Error[1164].CreateEx(TC_Events.Error.Error1164,FALSE,0);
Error[1165].CreateEx(TC_Events.Error.Error1165,FALSE,0);
Error[1166].CreateEx(TC_Events.Error.Error1166,FALSE,0);
Error[1167].CreateEx(TC_Events.Error.Error1167,FALSE,0);
Error[1168].CreateEx(TC_Events.Error.Error1168,FALSE,0);
Error[1169].CreateEx(TC_Events.Error.Error1169,FALSE,0);
Error[1170].CreateEx(TC_Events.Error.Error1170,FALSE,0);
Error[1171].CreateEx(TC_Events.Error.Error1171,FALSE,0);
Error[1172].CreateEx(TC_Events.Error.Error1172,FALSE,0);
Error[1173].CreateEx(TC_Events.Error.Error1173,FALSE,0);
Error[1174].CreateEx(TC_Events.Error.Error1174,FALSE,0);
Error[1175].CreateEx(TC_Events.Error.Error1175,FALSE,0);
Error[1176].CreateEx(TC_Events.Error.Error1176,FALSE,0);
Error[1177].CreateEx(TC_Events.Error.Error1177,FALSE,0);
Error[1178].CreateEx(TC_Events.Error.Error1178,FALSE,0);
Error[1179].CreateEx(TC_Events.Error.Error1179,FALSE,0);
Error[1180].CreateEx(TC_Events.Error.Error1180,FALSE,0);
Error[1181].CreateEx(TC_Events.Error.Error1181,FALSE,0);
Error[1182].CreateEx(TC_Events.Error.Error1182,FALSE,0);
Error[1183].CreateEx(TC_Events.Error.Error1183,FALSE,0);
Error[1184].CreateEx(TC_Events.Error.Error1184,FALSE,0);
Error[1185].CreateEx(TC_Events.Error.Error1185,FALSE,0);
Error[1186].CreateEx(TC_Events.Error.Error1186,FALSE,0);
Error[1187].CreateEx(TC_Events.Error.Error1187,FALSE,0);
Error[1188].CreateEx(TC_Events.Error.Error1188,FALSE,0);
Error[1189].CreateEx(TC_Events.Error.Error1189,FALSE,0);
Error[1190].CreateEx(TC_Events.Error.Error1190,FALSE,0);
Error[1191].CreateEx(TC_Events.Error.Error1191,FALSE,0);
Error[1192].CreateEx(TC_Events.Error.Error1192,FALSE,0);
Error[1193].CreateEx(TC_Events.Error.Error1193,FALSE,0);
Error[1194].CreateEx(TC_Events.Error.Error1194,FALSE,0);
Error[1195].CreateEx(TC_Events.Error.Error1195,FALSE,0);
Error[1196].CreateEx(TC_Events.Error.Error1196,FALSE,0);
Error[1197].CreateEx(TC_Events.Error.Error1197,FALSE,0);
Error[1198].CreateEx(TC_Events.Error.Error1198,FALSE,0);
Error[1199].CreateEx(TC_Events.Error.Error1199,FALSE,0);
Error[1200].CreateEx(TC_Events.Error.Error1200,FALSE,0);
Error[1201].CreateEx(TC_Events.Error.Error1201,FALSE,0);
Error[1202].CreateEx(TC_Events.Error.Error1202,FALSE,0);
Error[1203].CreateEx(TC_Events.Error.Error1203,FALSE,0);
Error[1204].CreateEx(TC_Events.Error.Error1204,FALSE,0);
Error[1205].CreateEx(TC_Events.Error.Error1205,FALSE,0);
Error[1206].CreateEx(TC_Events.Error.Error1206,FALSE,0);
Error[1207].CreateEx(TC_Events.Error.Error1207,FALSE,0);
Error[1208].CreateEx(TC_Events.Error.Error1208,FALSE,0);
Error[1209].CreateEx(TC_Events.Error.Error1209,FALSE,0);
Error[1210].CreateEx(TC_Events.Error.Error1210,FALSE,0);
Error[1211].CreateEx(TC_Events.Error.Error1211,FALSE,0);
Error[1212].CreateEx(TC_Events.Error.Error1212,FALSE,0);
Error[1213].CreateEx(TC_Events.Error.Error1213,FALSE,0);
Error[1214].CreateEx(TC_Events.Error.Error1214,FALSE,0);
Error[1215].CreateEx(TC_Events.Error.Error1215,FALSE,0);
Error[1216].CreateEx(TC_Events.Error.Error1216,FALSE,0);
Error[1217].CreateEx(TC_Events.Error.Error1217,FALSE,0);
Error[1218].CreateEx(TC_Events.Error.Error1218,FALSE,0);
Error[1219].CreateEx(TC_Events.Error.Error1219,FALSE,0);
Error[1220].CreateEx(TC_Events.Error.Error1220,FALSE,0);
Error[1221].CreateEx(TC_Events.Error.Error1221,FALSE,0);
Error[1222].CreateEx(TC_Events.Error.Error1222,FALSE,0);
Error[1223].CreateEx(TC_Events.Error.Error1223,FALSE,0);
Error[1224].CreateEx(TC_Events.Error.Error1224,FALSE,0);
Error[1225].CreateEx(TC_Events.Error.Error1225,FALSE,0);
Error[1226].CreateEx(TC_Events.Error.Error1226,FALSE,0);
Error[1227].CreateEx(TC_Events.Error.Error1227,FALSE,0);
Error[1228].CreateEx(TC_Events.Error.Error1228,FALSE,0);
Error[1229].CreateEx(TC_Events.Error.Error1229,FALSE,0);
Error[1230].CreateEx(TC_Events.Error.Error1230,FALSE,0);
Error[1231].CreateEx(TC_Events.Error.Error1231,FALSE,0);
Error[1232].CreateEx(TC_Events.Error.Error1232,FALSE,0);
Error[1233].CreateEx(TC_Events.Error.Error1233,FALSE,0);
Error[1234].CreateEx(TC_Events.Error.Error1234,FALSE,0);
Error[1235].CreateEx(TC_Events.Error.Error1235,FALSE,0);
Error[1236].CreateEx(TC_Events.Error.Error1236,FALSE,0);
Error[1237].CreateEx(TC_Events.Error.Error1237,FALSE,0);
Error[1238].CreateEx(TC_Events.Error.Error1238,FALSE,0);
Error[1239].CreateEx(TC_Events.Error.Error1239,FALSE,0);
Error[1240].CreateEx(TC_Events.Error.Error1240,FALSE,0);
Error[1241].CreateEx(TC_Events.Error.Error1241,FALSE,0);
Error[1242].CreateEx(TC_Events.Error.Error1242,FALSE,0);
Error[1243].CreateEx(TC_Events.Error.Error1243,FALSE,0);
Error[1244].CreateEx(TC_Events.Error.Error1244,FALSE,0);
Error[1245].CreateEx(TC_Events.Error.Error1245,FALSE,0);
Error[1246].CreateEx(TC_Events.Error.Error1246,FALSE,0);
Error[1247].CreateEx(TC_Events.Error.Error1247,FALSE,0);
Error[1248].CreateEx(TC_Events.Error.Error1248,FALSE,0);
Error[1249].CreateEx(TC_Events.Error.Error1249,FALSE,0);
Error[1250].CreateEx(TC_Events.Error.Error1250,FALSE,0);
Error[1251].CreateEx(TC_Events.Error.Error1251,FALSE,0);
Error[1252].CreateEx(TC_Events.Error.Error1252,FALSE,0);
Error[1253].CreateEx(TC_Events.Error.Error1253,FALSE,0);
Error[1254].CreateEx(TC_Events.Error.Error1254,FALSE,0);
Error[1255].CreateEx(TC_Events.Error.Error1255,FALSE,0);
Error[1256].CreateEx(TC_Events.Error.Error1256,FALSE,0);
Error[1257].CreateEx(TC_Events.Error.Error1257,FALSE,0);
Error[1258].CreateEx(TC_Events.Error.Error1258,FALSE,0);
Error[1259].CreateEx(TC_Events.Error.Error1259,FALSE,0);
Error[1260].CreateEx(TC_Events.Error.Error1260,FALSE,0);
Error[1261].CreateEx(TC_Events.Error.Error1261,FALSE,0);
Error[1262].CreateEx(TC_Events.Error.Error1262,FALSE,0);
Error[1263].CreateEx(TC_Events.Error.Error1263,FALSE,0);
Error[1264].CreateEx(TC_Events.Error.Error1264,FALSE,0);
Error[1265].CreateEx(TC_Events.Error.Error1265,FALSE,0);
Error[1266].CreateEx(TC_Events.Error.Error1266,FALSE,0);
Error[1267].CreateEx(TC_Events.Error.Error1267,FALSE,0);
Error[1268].CreateEx(TC_Events.Error.Error1268,FALSE,0);
Error[1269].CreateEx(TC_Events.Error.Error1269,FALSE,0);
Error[1270].CreateEx(TC_Events.Error.Error1270,FALSE,0);
Error[1271].CreateEx(TC_Events.Error.Error1271,FALSE,0);
Error[1272].CreateEx(TC_Events.Error.Error1272,FALSE,0);
Error[1273].CreateEx(TC_Events.Error.Error1273,FALSE,0);
Error[1274].CreateEx(TC_Events.Error.Error1274,FALSE,0);
Error[1275].CreateEx(TC_Events.Error.Error1275,FALSE,0);
Error[1276].CreateEx(TC_Events.Error.Error1276,FALSE,0);
Error[1277].CreateEx(TC_Events.Error.Error1277,FALSE,0);
Error[1278].CreateEx(TC_Events.Error.Error1278,FALSE,0);
Error[1279].CreateEx(TC_Events.Error.Error1279,FALSE,0);
Error[1280].CreateEx(TC_Events.Error.Error1280,FALSE,0);
Error[1281].CreateEx(TC_Events.Error.Error1281,FALSE,0);
Error[1282].CreateEx(TC_Events.Error.Error1282,FALSE,0);
Error[1283].CreateEx(TC_Events.Error.Error1283,FALSE,0);
Error[1284].CreateEx(TC_Events.Error.Error1284,FALSE,0);
Error[1285].CreateEx(TC_Events.Error.Error1285,FALSE,0);
Error[1286].CreateEx(TC_Events.Error.Error1286,FALSE,0);
Error[1287].CreateEx(TC_Events.Error.Error1287,FALSE,0);
Error[1288].CreateEx(TC_Events.Error.Error1288,FALSE,0);
Error[1289].CreateEx(TC_Events.Error.Error1289,FALSE,0);
Error[1290].CreateEx(TC_Events.Error.Error1290,FALSE,0);
Error[1291].CreateEx(TC_Events.Error.Error1291,FALSE,0);
Error[1292].CreateEx(TC_Events.Error.Error1292,FALSE,0);
Error[1293].CreateEx(TC_Events.Error.Error1293,FALSE,0);
Error[1294].CreateEx(TC_Events.Error.Error1294,FALSE,0);
Error[1295].CreateEx(TC_Events.Error.Error1295,FALSE,0);
Error[1296].CreateEx(TC_Events.Error.Error1296,FALSE,0);
Error[1297].CreateEx(TC_Events.Error.Error1297,FALSE,0);
Error[1298].CreateEx(TC_Events.Error.Error1298,FALSE,0);
Error[1299].CreateEx(TC_Events.Error.Error1299,FALSE,0);
Error[1300].CreateEx(TC_Events.Error.Error1300,FALSE,0);
Error[1301].CreateEx(TC_Events.Error.Error1301,FALSE,0);
Error[1302].CreateEx(TC_Events.Error.Error1302,FALSE,0);
Error[1303].CreateEx(TC_Events.Error.Error1303,FALSE,0);
Error[1304].CreateEx(TC_Events.Error.Error1304,FALSE,0);
Error[1305].CreateEx(TC_Events.Error.Error1305,FALSE,0);
Error[1306].CreateEx(TC_Events.Error.Error1306,FALSE,0);
Error[1307].CreateEx(TC_Events.Error.Error1307,FALSE,0);
Error[1308].CreateEx(TC_Events.Error.Error1308,FALSE,0);
Error[1309].CreateEx(TC_Events.Error.Error1309,FALSE,0);
Error[1310].CreateEx(TC_Events.Error.Error1310,FALSE,0);
Error[1311].CreateEx(TC_Events.Error.Error1311,FALSE,0);
Error[1312].CreateEx(TC_Events.Error.Error1312,FALSE,0);
Error[1313].CreateEx(TC_Events.Error.Error1313,FALSE,0);
Error[1314].CreateEx(TC_Events.Error.Error1314,FALSE,0);
Error[1315].CreateEx(TC_Events.Error.Error1315,FALSE,0);
Error[1316].CreateEx(TC_Events.Error.Error1316,FALSE,0);
Error[1317].CreateEx(TC_Events.Error.Error1317,FALSE,0);
Error[1318].CreateEx(TC_Events.Error.Error1318,FALSE,0);
Error[1319].CreateEx(TC_Events.Error.Error1319,FALSE,0);
Error[1320].CreateEx(TC_Events.Error.Error1320,FALSE,0);
Error[1321].CreateEx(TC_Events.Error.Error1321,FALSE,0);
Error[1322].CreateEx(TC_Events.Error.Error1322,FALSE,0);
Error[1323].CreateEx(TC_Events.Error.Error1323,FALSE,0);
Error[1324].CreateEx(TC_Events.Error.Error1324,FALSE,0);
Error[1325].CreateEx(TC_Events.Error.Error1325,FALSE,0);
Error[1326].CreateEx(TC_Events.Error.Error1326,FALSE,0);
Error[1327].CreateEx(TC_Events.Error.Error1327,FALSE,0);
Error[1328].CreateEx(TC_Events.Error.Error1328,FALSE,0);
Error[1329].CreateEx(TC_Events.Error.Error1329,FALSE,0);
Error[1330].CreateEx(TC_Events.Error.Error1330,FALSE,0);
Error[1331].CreateEx(TC_Events.Error.Error1331,FALSE,0);
Error[1332].CreateEx(TC_Events.Error.Error1332,FALSE,0);
Error[1333].CreateEx(TC_Events.Error.Error1333,FALSE,0);
Error[1334].CreateEx(TC_Events.Error.Error1334,FALSE,0);
Error[1335].CreateEx(TC_Events.Error.Error1335,FALSE,0);
Error[1336].CreateEx(TC_Events.Error.Error1336,FALSE,0);
Error[1337].CreateEx(TC_Events.Error.Error1337,FALSE,0);
Error[1338].CreateEx(TC_Events.Error.Error1338,FALSE,0);
Error[1339].CreateEx(TC_Events.Error.Error1339,FALSE,0);
Error[1340].CreateEx(TC_Events.Error.Error1340,FALSE,0);
Error[1341].CreateEx(TC_Events.Error.Error1341,FALSE,0);
Error[1342].CreateEx(TC_Events.Error.Error1342,FALSE,0);
Error[1343].CreateEx(TC_Events.Error.Error1343,FALSE,0);
Error[1344].CreateEx(TC_Events.Error.Error1344,FALSE,0);
Error[1345].CreateEx(TC_Events.Error.Error1345,FALSE,0);
Error[1346].CreateEx(TC_Events.Error.Error1346,FALSE,0);
Error[1347].CreateEx(TC_Events.Error.Error1347,FALSE,0);
Error[1348].CreateEx(TC_Events.Error.Error1348,FALSE,0);
Error[1349].CreateEx(TC_Events.Error.Error1349,FALSE,0);
Error[1350].CreateEx(TC_Events.Error.Error1350,FALSE,0);
Error[1351].CreateEx(TC_Events.Error.Error1351,FALSE,0);
Error[1352].CreateEx(TC_Events.Error.Error1352,FALSE,0);
Error[1353].CreateEx(TC_Events.Error.Error1353,FALSE,0);
Error[1354].CreateEx(TC_Events.Error.Error1354,FALSE,0);
Error[1355].CreateEx(TC_Events.Error.Error1355,FALSE,0);
Error[1356].CreateEx(TC_Events.Error.Error1356,FALSE,0);
Error[1357].CreateEx(TC_Events.Error.Error1357,FALSE,0);
Error[1358].CreateEx(TC_Events.Error.Error1358,FALSE,0);
Error[1359].CreateEx(TC_Events.Error.Error1359,FALSE,0);
Error[1360].CreateEx(TC_Events.Error.Error1360,FALSE,0);
Error[1361].CreateEx(TC_Events.Error.Error1361,FALSE,0);
Error[1362].CreateEx(TC_Events.Error.Error1362,FALSE,0);
Error[1363].CreateEx(TC_Events.Error.Error1363,FALSE,0);
Error[1364].CreateEx(TC_Events.Error.Error1364,FALSE,0);
Error[1365].CreateEx(TC_Events.Error.Error1365,FALSE,0);
Error[1366].CreateEx(TC_Events.Error.Error1366,FALSE,0);
Error[1367].CreateEx(TC_Events.Error.Error1367,FALSE,0);
Error[1368].CreateEx(TC_Events.Error.Error1368,FALSE,0);
Error[1369].CreateEx(TC_Events.Error.Error1369,FALSE,0);
Error[1370].CreateEx(TC_Events.Error.Error1370,FALSE,0);
Error[1371].CreateEx(TC_Events.Error.Error1371,FALSE,0);
Error[1372].CreateEx(TC_Events.Error.Error1372,FALSE,0);
Error[1373].CreateEx(TC_Events.Error.Error1373,FALSE,0);
Error[1374].CreateEx(TC_Events.Error.Error1374,FALSE,0);
Error[1375].CreateEx(TC_Events.Error.Error1375,FALSE,0);
Error[1376].CreateEx(TC_Events.Error.Error1376,FALSE,0);
Error[1377].CreateEx(TC_Events.Error.Error1377,FALSE,0);
Error[1378].CreateEx(TC_Events.Error.Error1378,FALSE,0);
Error[1379].CreateEx(TC_Events.Error.Error1379,FALSE,0);
Error[1380].CreateEx(TC_Events.Error.Error1380,FALSE,0);
Error[1381].CreateEx(TC_Events.Error.Error1381,FALSE,0);
Error[1382].CreateEx(TC_Events.Error.Error1382,FALSE,0);
Error[1383].CreateEx(TC_Events.Error.Error1383,FALSE,0);
Error[1384].CreateEx(TC_Events.Error.Error1384,FALSE,0);
Error[1385].CreateEx(TC_Events.Error.Error1385,FALSE,0);
Error[1386].CreateEx(TC_Events.Error.Error1386,FALSE,0);
Error[1387].CreateEx(TC_Events.Error.Error1387,FALSE,0);
Error[1388].CreateEx(TC_Events.Error.Error1388,FALSE,0);
Error[1389].CreateEx(TC_Events.Error.Error1389,FALSE,0);
Error[1390].CreateEx(TC_Events.Error.Error1390,FALSE,0);
Error[1391].CreateEx(TC_Events.Error.Error1391,FALSE,0);
Error[1392].CreateEx(TC_Events.Error.Error1392,FALSE,0);
Error[1393].CreateEx(TC_Events.Error.Error1393,FALSE,0);
Error[1394].CreateEx(TC_Events.Error.Error1394,FALSE,0);
Error[1395].CreateEx(TC_Events.Error.Error1395,FALSE,0);
Error[1396].CreateEx(TC_Events.Error.Error1396,FALSE,0);
Error[1397].CreateEx(TC_Events.Error.Error1397,FALSE,0);
Error[1398].CreateEx(TC_Events.Error.Error1398,FALSE,0);
Error[1399].CreateEx(TC_Events.Error.Error1399,FALSE,0);
Error[1400].CreateEx(TC_Events.Error.Error1400,FALSE,0);
Error[1401].CreateEx(TC_Events.Error.Error1401,FALSE,0);
Error[1402].CreateEx(TC_Events.Error.Error1402,FALSE,0);
Error[1403].CreateEx(TC_Events.Error.Error1403,FALSE,0);
Error[1404].CreateEx(TC_Events.Error.Error1404,FALSE,0);
Error[1405].CreateEx(TC_Events.Error.Error1405,FALSE,0);
Error[1406].CreateEx(TC_Events.Error.Error1406,FALSE,0);
Error[1407].CreateEx(TC_Events.Error.Error1407,FALSE,0);
Error[1408].CreateEx(TC_Events.Error.Error1408,FALSE,0);
Error[1409].CreateEx(TC_Events.Error.Error1409,FALSE,0);
Error[1410].CreateEx(TC_Events.Error.Error1410,FALSE,0);
Error[1411].CreateEx(TC_Events.Error.Error1411,FALSE,0);
Error[1412].CreateEx(TC_Events.Error.Error1412,FALSE,0);
Error[1413].CreateEx(TC_Events.Error.Error1413,FALSE,0);
Error[1414].CreateEx(TC_Events.Error.Error1414,FALSE,0);
Error[1415].CreateEx(TC_Events.Error.Error1415,FALSE,0);
Error[1416].CreateEx(TC_Events.Error.Error1416,FALSE,0);
Error[1417].CreateEx(TC_Events.Error.Error1417,FALSE,0);
Error[1418].CreateEx(TC_Events.Error.Error1418,FALSE,0);
Error[1419].CreateEx(TC_Events.Error.Error1419,FALSE,0);
Error[1420].CreateEx(TC_Events.Error.Error1420,FALSE,0);
Error[1421].CreateEx(TC_Events.Error.Error1421,FALSE,0);
Error[1422].CreateEx(TC_Events.Error.Error1422,FALSE,0);
Error[1423].CreateEx(TC_Events.Error.Error1423,FALSE,0);
Error[1424].CreateEx(TC_Events.Error.Error1424,FALSE,0);
Error[1425].CreateEx(TC_Events.Error.Error1425,FALSE,0);
Error[1426].CreateEx(TC_Events.Error.Error1426,FALSE,0);
Error[1427].CreateEx(TC_Events.Error.Error1427,FALSE,0);
Error[1428].CreateEx(TC_Events.Error.Error1428,FALSE,0);
Error[1429].CreateEx(TC_Events.Error.Error1429,FALSE,0);
Error[1430].CreateEx(TC_Events.Error.Error1430,FALSE,0);
Error[1431].CreateEx(TC_Events.Error.Error1431,FALSE,0);
Error[1432].CreateEx(TC_Events.Error.Error1432,FALSE,0);
Error[1433].CreateEx(TC_Events.Error.Error1433,FALSE,0);
Error[1434].CreateEx(TC_Events.Error.Error1434,FALSE,0);
Error[1435].CreateEx(TC_Events.Error.Error1435,FALSE,0);
Error[1436].CreateEx(TC_Events.Error.Error1436,FALSE,0);
Error[1437].CreateEx(TC_Events.Error.Error1437,FALSE,0);
Error[1438].CreateEx(TC_Events.Error.Error1438,FALSE,0);
Error[1439].CreateEx(TC_Events.Error.Error1439,FALSE,0);
Error[1440].CreateEx(TC_Events.Error.Error1440,FALSE,0);
Error[1441].CreateEx(TC_Events.Error.Error1441,FALSE,0);
Error[1442].CreateEx(TC_Events.Error.Error1442,FALSE,0);
Error[1443].CreateEx(TC_Events.Error.Error1443,FALSE,0);
Error[1444].CreateEx(TC_Events.Error.Error1444,FALSE,0);
Error[1445].CreateEx(TC_Events.Error.Error1445,FALSE,0);
Error[1446].CreateEx(TC_Events.Error.Error1446,FALSE,0);
Error[1447].CreateEx(TC_Events.Error.Error1447,FALSE,0);
Error[1448].CreateEx(TC_Events.Error.Error1448,FALSE,0);
Error[1449].CreateEx(TC_Events.Error.Error1449,FALSE,0);
Error[1450].CreateEx(TC_Events.Error.Error1450,FALSE,0);
Error[1451].CreateEx(TC_Events.Error.Error1451,FALSE,0);
Error[1452].CreateEx(TC_Events.Error.Error1452,FALSE,0);
Error[1453].CreateEx(TC_Events.Error.Error1453,FALSE,0);
Error[1454].CreateEx(TC_Events.Error.Error1454,FALSE,0);
Error[1455].CreateEx(TC_Events.Error.Error1455,FALSE,0);
Error[1456].CreateEx(TC_Events.Error.Error1456,FALSE,0);
Error[1457].CreateEx(TC_Events.Error.Error1457,FALSE,0);
Error[1458].CreateEx(TC_Events.Error.Error1458,FALSE,0);
Error[1459].CreateEx(TC_Events.Error.Error1459,FALSE,0);
Error[1460].CreateEx(TC_Events.Error.Error1460,FALSE,0);
Error[1461].CreateEx(TC_Events.Error.Error1461,FALSE,0);
Error[1462].CreateEx(TC_Events.Error.Error1462,FALSE,0);
Error[1463].CreateEx(TC_Events.Error.Error1463,FALSE,0);
Error[1464].CreateEx(TC_Events.Error.Error1464,FALSE,0);
Error[1465].CreateEx(TC_Events.Error.Error1465,FALSE,0);
Error[1466].CreateEx(TC_Events.Error.Error1466,FALSE,0);
Error[1467].CreateEx(TC_Events.Error.Error1467,FALSE,0);
Error[1468].CreateEx(TC_Events.Error.Error1468,FALSE,0);
Error[1469].CreateEx(TC_Events.Error.Error1469,FALSE,0);
Error[1470].CreateEx(TC_Events.Error.Error1470,FALSE,0);
Error[1471].CreateEx(TC_Events.Error.Error1471,FALSE,0);
Error[1472].CreateEx(TC_Events.Error.Error1472,FALSE,0);
Error[1473].CreateEx(TC_Events.Error.Error1473,FALSE,0);
Error[1474].CreateEx(TC_Events.Error.Error1474,FALSE,0);
Error[1475].CreateEx(TC_Events.Error.Error1475,FALSE,0);
Error[1476].CreateEx(TC_Events.Error.Error1476,FALSE,0);
Error[1477].CreateEx(TC_Events.Error.Error1477,FALSE,0);
Error[1478].CreateEx(TC_Events.Error.Error1478,FALSE,0);
Error[1479].CreateEx(TC_Events.Error.Error1479,FALSE,0);
Error[1480].CreateEx(TC_Events.Error.Error1480,FALSE,0);
Error[1481].CreateEx(TC_Events.Error.Error1481,FALSE,0);
Error[1482].CreateEx(TC_Events.Error.Error1482,FALSE,0);
Error[1483].CreateEx(TC_Events.Error.Error1483,FALSE,0);
Error[1484].CreateEx(TC_Events.Error.Error1484,FALSE,0);
Error[1485].CreateEx(TC_Events.Error.Error1485,FALSE,0);
Error[1486].CreateEx(TC_Events.Error.Error1486,FALSE,0);
Error[1487].CreateEx(TC_Events.Error.Error1487,FALSE,0);
Error[1488].CreateEx(TC_Events.Error.Error1488,FALSE,0);
Error[1489].CreateEx(TC_Events.Error.Error1489,FALSE,0);
Error[1490].CreateEx(TC_Events.Error.Error1490,FALSE,0);
Error[1491].CreateEx(TC_Events.Error.Error1491,FALSE,0);
Error[1492].CreateEx(TC_Events.Error.Error1492,FALSE,0);
Error[1493].CreateEx(TC_Events.Error.Error1493,FALSE,0);
Error[1494].CreateEx(TC_Events.Error.Error1494,FALSE,0);
Error[1495].CreateEx(TC_Events.Error.Error1495,FALSE,0);
Error[1496].CreateEx(TC_Events.Error.Error1496,FALSE,0);
Error[1497].CreateEx(TC_Events.Error.Error1497,FALSE,0);
Error[1498].CreateEx(TC_Events.Error.Error1498,FALSE,0);
Error[1499].CreateEx(TC_Events.Error.Error1499,FALSE,0);
Error[1500].CreateEx(TC_Events.Error.Error1500,FALSE,0);
Error[1501].CreateEx(TC_Events.Error.Error1501,FALSE,0);
Error[1502].CreateEx(TC_Events.Error.Error1502,FALSE,0);
Error[1503].CreateEx(TC_Events.Error.Error1503,FALSE,0);
Error[1504].CreateEx(TC_Events.Error.Error1504,FALSE,0);
Error[1505].CreateEx(TC_Events.Error.Error1505,FALSE,0);
Error[1506].CreateEx(TC_Events.Error.Error1506,FALSE,0);
Error[1507].CreateEx(TC_Events.Error.Error1507,FALSE,0);
Error[1508].CreateEx(TC_Events.Error.Error1508,FALSE,0);
Error[1509].CreateEx(TC_Events.Error.Error1509,FALSE,0);
Error[1510].CreateEx(TC_Events.Error.Error1510,FALSE,0);
Error[1511].CreateEx(TC_Events.Error.Error1511,FALSE,0);
Error[1512].CreateEx(TC_Events.Error.Error1512,FALSE,0);
Error[1513].CreateEx(TC_Events.Error.Error1513,FALSE,0);
Error[1514].CreateEx(TC_Events.Error.Error1514,FALSE,0);
Error[1515].CreateEx(TC_Events.Error.Error1515,FALSE,0);
Error[1516].CreateEx(TC_Events.Error.Error1516,FALSE,0);
Error[1517].CreateEx(TC_Events.Error.Error1517,FALSE,0);
Error[1518].CreateEx(TC_Events.Error.Error1518,FALSE,0);
Error[1519].CreateEx(TC_Events.Error.Error1519,FALSE,0);
Error[1520].CreateEx(TC_Events.Error.Error1520,FALSE,0);
Error[1521].CreateEx(TC_Events.Error.Error1521,FALSE,0);
Error[1522].CreateEx(TC_Events.Error.Error1522,FALSE,0);
Error[1523].CreateEx(TC_Events.Error.Error1523,FALSE,0);
Error[1524].CreateEx(TC_Events.Error.Error1524,FALSE,0);
Error[1525].CreateEx(TC_Events.Error.Error1525,FALSE,0);
Error[1526].CreateEx(TC_Events.Error.Error1526,FALSE,0);
Error[1527].CreateEx(TC_Events.Error.Error1527,FALSE,0);
Error[1528].CreateEx(TC_Events.Error.Error1528,FALSE,0);
Error[1529].CreateEx(TC_Events.Error.Error1529,FALSE,0);
Error[1530].CreateEx(TC_Events.Error.Error1530,FALSE,0);
Error[1531].CreateEx(TC_Events.Error.Error1531,FALSE,0);
Error[1532].CreateEx(TC_Events.Error.Error1532,FALSE,0);
Error[1533].CreateEx(TC_Events.Error.Error1533,FALSE,0);
Error[1534].CreateEx(TC_Events.Error.Error1534,FALSE,0);
Error[1535].CreateEx(TC_Events.Error.Error1535,FALSE,0);
Error[1536].CreateEx(TC_Events.Error.Error1536,FALSE,0);
Error[1537].CreateEx(TC_Events.Error.Error1537,FALSE,0);
Error[1538].CreateEx(TC_Events.Error.Error1538,FALSE,0);
Error[1539].CreateEx(TC_Events.Error.Error1539,FALSE,0);
Error[1540].CreateEx(TC_Events.Error.Error1540,FALSE,0);
Error[1541].CreateEx(TC_Events.Error.Error1541,FALSE,0);
Error[1542].CreateEx(TC_Events.Error.Error1542,FALSE,0);
Error[1543].CreateEx(TC_Events.Error.Error1543,FALSE,0);
Error[1544].CreateEx(TC_Events.Error.Error1544,FALSE,0);
Error[1545].CreateEx(TC_Events.Error.Error1545,FALSE,0);
Error[1546].CreateEx(TC_Events.Error.Error1546,FALSE,0);
Error[1547].CreateEx(TC_Events.Error.Error1547,FALSE,0);
Error[1548].CreateEx(TC_Events.Error.Error1548,FALSE,0);
Error[1549].CreateEx(TC_Events.Error.Error1549,FALSE,0);
Error[1550].CreateEx(TC_Events.Error.Error1550,FALSE,0);
Error[1551].CreateEx(TC_Events.Error.Error1551,FALSE,0);
Error[1552].CreateEx(TC_Events.Error.Error1552,FALSE,0);
Error[1553].CreateEx(TC_Events.Error.Error1553,FALSE,0);
Error[1554].CreateEx(TC_Events.Error.Error1554,FALSE,0);
Error[1555].CreateEx(TC_Events.Error.Error1555,FALSE,0);
Error[1556].CreateEx(TC_Events.Error.Error1556,FALSE,0);
Error[1557].CreateEx(TC_Events.Error.Error1557,FALSE,0);
Error[1558].CreateEx(TC_Events.Error.Error1558,FALSE,0);
Error[1559].CreateEx(TC_Events.Error.Error1559,FALSE,0);
Error[1560].CreateEx(TC_Events.Error.Error1560,FALSE,0);
Error[1561].CreateEx(TC_Events.Error.Error1561,FALSE,0);
Error[1562].CreateEx(TC_Events.Error.Error1562,FALSE,0);
Error[1563].CreateEx(TC_Events.Error.Error1563,FALSE,0);
Error[1564].CreateEx(TC_Events.Error.Error1564,FALSE,0);
Error[1565].CreateEx(TC_Events.Error.Error1565,FALSE,0);
Error[1566].CreateEx(TC_Events.Error.Error1566,FALSE,0);
Error[1567].CreateEx(TC_Events.Error.Error1567,FALSE,0);
Error[1568].CreateEx(TC_Events.Error.Error1568,FALSE,0);
Error[1569].CreateEx(TC_Events.Error.Error1569,FALSE,0);
Error[1570].CreateEx(TC_Events.Error.Error1570,FALSE,0);
Error[1571].CreateEx(TC_Events.Error.Error1571,FALSE,0);
Error[1572].CreateEx(TC_Events.Error.Error1572,FALSE,0);
Error[1573].CreateEx(TC_Events.Error.Error1573,FALSE,0);
Error[1574].CreateEx(TC_Events.Error.Error1574,FALSE,0);
Error[1575].CreateEx(TC_Events.Error.Error1575,FALSE,0);
Error[1576].CreateEx(TC_Events.Error.Error1576,FALSE,0);
Error[1577].CreateEx(TC_Events.Error.Error1577,FALSE,0);
Error[1578].CreateEx(TC_Events.Error.Error1578,FALSE,0);
Error[1579].CreateEx(TC_Events.Error.Error1579,FALSE,0);
Error[1580].CreateEx(TC_Events.Error.Error1580,FALSE,0);
Error[1581].CreateEx(TC_Events.Error.Error1581,FALSE,0);
Error[1582].CreateEx(TC_Events.Error.Error1582,FALSE,0);
Error[1583].CreateEx(TC_Events.Error.Error1583,FALSE,0);
Error[1584].CreateEx(TC_Events.Error.Error1584,FALSE,0);
Error[1585].CreateEx(TC_Events.Error.Error1585,FALSE,0);
Error[1586].CreateEx(TC_Events.Error.Error1586,FALSE,0);
Error[1587].CreateEx(TC_Events.Error.Error1587,FALSE,0);
Error[1588].CreateEx(TC_Events.Error.Error1588,FALSE,0);
Error[1589].CreateEx(TC_Events.Error.Error1589,FALSE,0);
Error[1590].CreateEx(TC_Events.Error.Error1590,FALSE,0);
Error[1591].CreateEx(TC_Events.Error.Error1591,FALSE,0);
Error[1592].CreateEx(TC_Events.Error.Error1592,FALSE,0);
Error[1593].CreateEx(TC_Events.Error.Error1593,FALSE,0);
Error[1594].CreateEx(TC_Events.Error.Error1594,FALSE,0);
Error[1595].CreateEx(TC_Events.Error.Error1595,FALSE,0);
Error[1596].CreateEx(TC_Events.Error.Error1596,FALSE,0);
Error[1597].CreateEx(TC_Events.Error.Error1597,FALSE,0);
Error[1598].CreateEx(TC_Events.Error.Error1598,FALSE,0);
Error[1599].CreateEx(TC_Events.Error.Error1599,FALSE,0);
Error[1600].CreateEx(TC_Events.Error.Error1600,FALSE,0);
Error[1601].CreateEx(TC_Events.Error.Error1601,FALSE,0);
Error[1602].CreateEx(TC_Events.Error.Error1602,FALSE,0);
Error[1603].CreateEx(TC_Events.Error.Error1603,FALSE,0);
Error[1604].CreateEx(TC_Events.Error.Error1604,FALSE,0);
Error[1605].CreateEx(TC_Events.Error.Error1605,FALSE,0);
Error[1606].CreateEx(TC_Events.Error.Error1606,FALSE,0);
Error[1607].CreateEx(TC_Events.Error.Error1607,FALSE,0);
Error[1608].CreateEx(TC_Events.Error.Error1608,FALSE,0);
Error[1609].CreateEx(TC_Events.Error.Error1609,FALSE,0);
Error[1610].CreateEx(TC_Events.Error.Error1610,FALSE,0);
Error[1611].CreateEx(TC_Events.Error.Error1611,FALSE,0);
Error[1612].CreateEx(TC_Events.Error.Error1612,FALSE,0);
Error[1613].CreateEx(TC_Events.Error.Error1613,FALSE,0);
Error[1614].CreateEx(TC_Events.Error.Error1614,FALSE,0);
Error[1615].CreateEx(TC_Events.Error.Error1615,FALSE,0);
Error[1616].CreateEx(TC_Events.Error.Error1616,FALSE,0);
Error[1617].CreateEx(TC_Events.Error.Error1617,FALSE,0);
Error[1618].CreateEx(TC_Events.Error.Error1618,FALSE,0);
Error[1619].CreateEx(TC_Events.Error.Error1619,FALSE,0);
Error[1620].CreateEx(TC_Events.Error.Error1620,FALSE,0);
Error[1621].CreateEx(TC_Events.Error.Error1621,FALSE,0);
Error[1622].CreateEx(TC_Events.Error.Error1622,FALSE,0);
Error[1623].CreateEx(TC_Events.Error.Error1623,FALSE,0);
Error[1624].CreateEx(TC_Events.Error.Error1624,FALSE,0);
Error[1625].CreateEx(TC_Events.Error.Error1625,FALSE,0);
Error[1626].CreateEx(TC_Events.Error.Error1626,FALSE,0);
Error[1627].CreateEx(TC_Events.Error.Error1627,FALSE,0);
Error[1628].CreateEx(TC_Events.Error.Error1628,FALSE,0);
Error[1629].CreateEx(TC_Events.Error.Error1629,FALSE,0);
Error[1630].CreateEx(TC_Events.Error.Error1630,FALSE,0);
Error[1631].CreateEx(TC_Events.Error.Error1631,FALSE,0);
Error[1632].CreateEx(TC_Events.Error.Error1632,FALSE,0);
Error[1633].CreateEx(TC_Events.Error.Error1633,FALSE,0);
Error[1634].CreateEx(TC_Events.Error.Error1634,FALSE,0);
Error[1635].CreateEx(TC_Events.Error.Error1635,FALSE,0);
Error[1636].CreateEx(TC_Events.Error.Error1636,FALSE,0);
Error[1637].CreateEx(TC_Events.Error.Error1637,FALSE,0);
Error[1638].CreateEx(TC_Events.Error.Error1638,FALSE,0);
Error[1639].CreateEx(TC_Events.Error.Error1639,FALSE,0);
Error[1640].CreateEx(TC_Events.Error.Error1640,FALSE,0);
Error[1641].CreateEx(TC_Events.Error.Error1641,FALSE,0);
Error[1642].CreateEx(TC_Events.Error.Error1642,FALSE,0);
Error[1643].CreateEx(TC_Events.Error.Error1643,FALSE,0);
Error[1644].CreateEx(TC_Events.Error.Error1644,FALSE,0);
Error[1645].CreateEx(TC_Events.Error.Error1645,FALSE,0);
Error[1646].CreateEx(TC_Events.Error.Error1646,FALSE,0);
Error[1647].CreateEx(TC_Events.Error.Error1647,FALSE,0);
Error[1648].CreateEx(TC_Events.Error.Error1648,FALSE,0);
Error[1649].CreateEx(TC_Events.Error.Error1649,FALSE,0);
Error[1650].CreateEx(TC_Events.Error.Error1650,FALSE,0);
Error[1651].CreateEx(TC_Events.Error.Error1651,FALSE,0);
Error[1652].CreateEx(TC_Events.Error.Error1652,FALSE,0);
Error[1653].CreateEx(TC_Events.Error.Error1653,FALSE,0);
Error[1654].CreateEx(TC_Events.Error.Error1654,FALSE,0);
Error[1655].CreateEx(TC_Events.Error.Error1655,FALSE,0);
Error[1656].CreateEx(TC_Events.Error.Error1656,FALSE,0);
Error[1657].CreateEx(TC_Events.Error.Error1657,FALSE,0);
Error[1658].CreateEx(TC_Events.Error.Error1658,FALSE,0);
Error[1659].CreateEx(TC_Events.Error.Error1659,FALSE,0);
Error[1660].CreateEx(TC_Events.Error.Error1660,FALSE,0);
Error[1661].CreateEx(TC_Events.Error.Error1661,FALSE,0);
Error[1662].CreateEx(TC_Events.Error.Error1662,FALSE,0);
Error[1663].CreateEx(TC_Events.Error.Error1663,FALSE,0);
Error[1664].CreateEx(TC_Events.Error.Error1664,FALSE,0);
Error[1665].CreateEx(TC_Events.Error.Error1665,FALSE,0);
Error[1666].CreateEx(TC_Events.Error.Error1666,FALSE,0);
Error[1667].CreateEx(TC_Events.Error.Error1667,FALSE,0);
Error[1668].CreateEx(TC_Events.Error.Error1668,FALSE,0);
Error[1669].CreateEx(TC_Events.Error.Error1669,FALSE,0);
Error[1670].CreateEx(TC_Events.Error.Error1670,FALSE,0);
Error[1671].CreateEx(TC_Events.Error.Error1671,FALSE,0);
Error[1672].CreateEx(TC_Events.Error.Error1672,FALSE,0);
Error[1673].CreateEx(TC_Events.Error.Error1673,FALSE,0);
Error[1674].CreateEx(TC_Events.Error.Error1674,FALSE,0);
Error[1675].CreateEx(TC_Events.Error.Error1675,FALSE,0);
Error[1676].CreateEx(TC_Events.Error.Error1676,FALSE,0);
Error[1677].CreateEx(TC_Events.Error.Error1677,FALSE,0);
Error[1678].CreateEx(TC_Events.Error.Error1678,FALSE,0);
Error[1679].CreateEx(TC_Events.Error.Error1679,FALSE,0);
Error[1680].CreateEx(TC_Events.Error.Error1680,FALSE,0);
Error[1681].CreateEx(TC_Events.Error.Error1681,FALSE,0);
Error[1682].CreateEx(TC_Events.Error.Error1682,FALSE,0);
Error[1683].CreateEx(TC_Events.Error.Error1683,FALSE,0);
Error[1684].CreateEx(TC_Events.Error.Error1684,FALSE,0);
Error[1685].CreateEx(TC_Events.Error.Error1685,FALSE,0);
Error[1686].CreateEx(TC_Events.Error.Error1686,FALSE,0);
Error[1687].CreateEx(TC_Events.Error.Error1687,FALSE,0);
Error[1688].CreateEx(TC_Events.Error.Error1688,FALSE,0);
Error[1689].CreateEx(TC_Events.Error.Error1689,FALSE,0);
Error[1690].CreateEx(TC_Events.Error.Error1690,FALSE,0);
Error[1691].CreateEx(TC_Events.Error.Error1691,FALSE,0);
Error[1692].CreateEx(TC_Events.Error.Error1692,FALSE,0);
Error[1693].CreateEx(TC_Events.Error.Error1693,FALSE,0);
Error[1694].CreateEx(TC_Events.Error.Error1694,FALSE,0);
Error[1695].CreateEx(TC_Events.Error.Error1695,FALSE,0);
Error[1696].CreateEx(TC_Events.Error.Error1696,FALSE,0);
Error[1697].CreateEx(TC_Events.Error.Error1697,FALSE,0);
Error[1698].CreateEx(TC_Events.Error.Error1698,FALSE,0);
Error[1699].CreateEx(TC_Events.Error.Error1699,FALSE,0);
Error[1700].CreateEx(TC_Events.Error.Error1700,FALSE,0);
Error[1701].CreateEx(TC_Events.Error.Error1701,FALSE,0);
Error[1702].CreateEx(TC_Events.Error.Error1702,FALSE,0);
Error[1703].CreateEx(TC_Events.Error.Error1703,FALSE,0);
Error[1704].CreateEx(TC_Events.Error.Error1704,FALSE,0);
Error[1705].CreateEx(TC_Events.Error.Error1705,FALSE,0);
Error[1706].CreateEx(TC_Events.Error.Error1706,FALSE,0);
Error[1707].CreateEx(TC_Events.Error.Error1707,FALSE,0);
Error[1708].CreateEx(TC_Events.Error.Error1708,FALSE,0);
Error[1709].CreateEx(TC_Events.Error.Error1709,FALSE,0);
Error[1710].CreateEx(TC_Events.Error.Error1710,FALSE,0);
Error[1711].CreateEx(TC_Events.Error.Error1711,FALSE,0);
Error[1712].CreateEx(TC_Events.Error.Error1712,FALSE,0);
Error[1713].CreateEx(TC_Events.Error.Error1713,FALSE,0);
Error[1714].CreateEx(TC_Events.Error.Error1714,FALSE,0);
Error[1715].CreateEx(TC_Events.Error.Error1715,FALSE,0);
Error[1716].CreateEx(TC_Events.Error.Error1716,FALSE,0);
Error[1717].CreateEx(TC_Events.Error.Error1717,FALSE,0);
Error[1718].CreateEx(TC_Events.Error.Error1718,FALSE,0);
Error[1719].CreateEx(TC_Events.Error.Error1719,FALSE,0);
Error[1720].CreateEx(TC_Events.Error.Error1720,FALSE,0);
Error[1721].CreateEx(TC_Events.Error.Error1721,FALSE,0);
Error[1722].CreateEx(TC_Events.Error.Error1722,FALSE,0);
Error[1723].CreateEx(TC_Events.Error.Error1723,FALSE,0);
Error[1724].CreateEx(TC_Events.Error.Error1724,FALSE,0);
Error[1725].CreateEx(TC_Events.Error.Error1725,FALSE,0);
Error[1726].CreateEx(TC_Events.Error.Error1726,FALSE,0);
Error[1727].CreateEx(TC_Events.Error.Error1727,FALSE,0);
Error[1728].CreateEx(TC_Events.Error.Error1728,FALSE,0);
Error[1729].CreateEx(TC_Events.Error.Error1729,FALSE,0);
Error[1730].CreateEx(TC_Events.Error.Error1730,FALSE,0);
Error[1731].CreateEx(TC_Events.Error.Error1731,FALSE,0);
Error[1732].CreateEx(TC_Events.Error.Error1732,FALSE,0);
Error[1733].CreateEx(TC_Events.Error.Error1733,FALSE,0);
Error[1734].CreateEx(TC_Events.Error.Error1734,FALSE,0);
Error[1735].CreateEx(TC_Events.Error.Error1735,FALSE,0);
Error[1736].CreateEx(TC_Events.Error.Error1736,FALSE,0);
Error[1737].CreateEx(TC_Events.Error.Error1737,FALSE,0);
Error[1738].CreateEx(TC_Events.Error.Error1738,FALSE,0);
Error[1739].CreateEx(TC_Events.Error.Error1739,FALSE,0);
Error[1740].CreateEx(TC_Events.Error.Error1740,FALSE,0);
Error[1741].CreateEx(TC_Events.Error.Error1741,FALSE,0);
Error[1742].CreateEx(TC_Events.Error.Error1742,FALSE,0);
Error[1743].CreateEx(TC_Events.Error.Error1743,FALSE,0);
Error[1744].CreateEx(TC_Events.Error.Error1744,FALSE,0);
Error[1745].CreateEx(TC_Events.Error.Error1745,FALSE,0);
Error[1746].CreateEx(TC_Events.Error.Error1746,FALSE,0);
Error[1747].CreateEx(TC_Events.Error.Error1747,FALSE,0);
Error[1748].CreateEx(TC_Events.Error.Error1748,FALSE,0);
Error[1749].CreateEx(TC_Events.Error.Error1749,FALSE,0);
Error[1750].CreateEx(TC_Events.Error.Error1750,FALSE,0);
Error[1751].CreateEx(TC_Events.Error.Error1751,FALSE,0);
Error[1752].CreateEx(TC_Events.Error.Error1752,FALSE,0);
Error[1753].CreateEx(TC_Events.Error.Error1753,FALSE,0);
Error[1754].CreateEx(TC_Events.Error.Error1754,FALSE,0);
Error[1755].CreateEx(TC_Events.Error.Error1755,FALSE,0);
Error[1756].CreateEx(TC_Events.Error.Error1756,FALSE,0);
Error[1757].CreateEx(TC_Events.Error.Error1757,FALSE,0);
Error[1758].CreateEx(TC_Events.Error.Error1758,FALSE,0);
Error[1759].CreateEx(TC_Events.Error.Error1759,FALSE,0);
Error[1760].CreateEx(TC_Events.Error.Error1760,FALSE,0);
Error[1761].CreateEx(TC_Events.Error.Error1761,FALSE,0);
Error[1762].CreateEx(TC_Events.Error.Error1762,FALSE,0);
Error[1763].CreateEx(TC_Events.Error.Error1763,FALSE,0);
Error[1764].CreateEx(TC_Events.Error.Error1764,FALSE,0);
Error[1765].CreateEx(TC_Events.Error.Error1765,FALSE,0);
Error[1766].CreateEx(TC_Events.Error.Error1766,FALSE,0);
Error[1767].CreateEx(TC_Events.Error.Error1767,FALSE,0);
Error[1768].CreateEx(TC_Events.Error.Error1768,FALSE,0);
Error[1769].CreateEx(TC_Events.Error.Error1769,FALSE,0);
Error[1770].CreateEx(TC_Events.Error.Error1770,FALSE,0);
Error[1771].CreateEx(TC_Events.Error.Error1771,FALSE,0);
Error[1772].CreateEx(TC_Events.Error.Error1772,FALSE,0);
Error[1773].CreateEx(TC_Events.Error.Error1773,FALSE,0);
Error[1774].CreateEx(TC_Events.Error.Error1774,FALSE,0);
Error[1775].CreateEx(TC_Events.Error.Error1775,FALSE,0);
Error[1776].CreateEx(TC_Events.Error.Error1776,FALSE,0);
Error[1777].CreateEx(TC_Events.Error.Error1777,FALSE,0);
Error[1778].CreateEx(TC_Events.Error.Error1778,FALSE,0);
Error[1779].CreateEx(TC_Events.Error.Error1779,FALSE,0);
Error[1780].CreateEx(TC_Events.Error.Error1780,FALSE,0);
Error[1781].CreateEx(TC_Events.Error.Error1781,FALSE,0);
Error[1782].CreateEx(TC_Events.Error.Error1782,FALSE,0);
Error[1783].CreateEx(TC_Events.Error.Error1783,FALSE,0);
Error[1784].CreateEx(TC_Events.Error.Error1784,FALSE,0);
Error[1785].CreateEx(TC_Events.Error.Error1785,FALSE,0);
Error[1786].CreateEx(TC_Events.Error.Error1786,FALSE,0);
Error[1787].CreateEx(TC_Events.Error.Error1787,FALSE,0);
Error[1788].CreateEx(TC_Events.Error.Error1788,FALSE,0);
Error[1789].CreateEx(TC_Events.Error.Error1789,FALSE,0);
Error[1790].CreateEx(TC_Events.Error.Error1790,FALSE,0);
Error[1791].CreateEx(TC_Events.Error.Error1791,FALSE,0);
Error[1792].CreateEx(TC_Events.Error.Error1792,FALSE,0);
Error[1793].CreateEx(TC_Events.Error.Error1793,FALSE,0);
Error[1794].CreateEx(TC_Events.Error.Error1794,FALSE,0);
Error[1795].CreateEx(TC_Events.Error.Error1795,FALSE,0);
Error[1796].CreateEx(TC_Events.Error.Error1796,FALSE,0);
Error[1797].CreateEx(TC_Events.Error.Error1797,FALSE,0);
Error[1798].CreateEx(TC_Events.Error.Error1798,FALSE,0);
Error[1799].CreateEx(TC_Events.Error.Error1799,FALSE,0);
Error[1800].CreateEx(TC_Events.Error.Error1800,FALSE,0);
Error[1801].CreateEx(TC_Events.Error.Error1801,FALSE,0);
Error[1802].CreateEx(TC_Events.Error.Error1802,FALSE,0);
Error[1803].CreateEx(TC_Events.Error.Error1803,FALSE,0);
Error[1804].CreateEx(TC_Events.Error.Error1804,FALSE,0);
Error[1805].CreateEx(TC_Events.Error.Error1805,FALSE,0);
Error[1806].CreateEx(TC_Events.Error.Error1806,FALSE,0);
Error[1807].CreateEx(TC_Events.Error.Error1807,FALSE,0);
Error[1808].CreateEx(TC_Events.Error.Error1808,FALSE,0);
Error[1809].CreateEx(TC_Events.Error.Error1809,FALSE,0);
Error[1810].CreateEx(TC_Events.Error.Error1810,FALSE,0);
Error[1811].CreateEx(TC_Events.Error.Error1811,FALSE,0);
Error[1812].CreateEx(TC_Events.Error.Error1812,FALSE,0);
Error[1813].CreateEx(TC_Events.Error.Error1813,FALSE,0);
Error[1814].CreateEx(TC_Events.Error.Error1814,FALSE,0);
Error[1815].CreateEx(TC_Events.Error.Error1815,FALSE,0);
Error[1816].CreateEx(TC_Events.Error.Error1816,FALSE,0);
Error[1817].CreateEx(TC_Events.Error.Error1817,FALSE,0);
Error[1818].CreateEx(TC_Events.Error.Error1818,FALSE,0);
Error[1819].CreateEx(TC_Events.Error.Error1819,FALSE,0);
Error[1820].CreateEx(TC_Events.Error.Error1820,FALSE,0);
Error[1821].CreateEx(TC_Events.Error.Error1821,FALSE,0);
Error[1822].CreateEx(TC_Events.Error.Error1822,FALSE,0);
Error[1823].CreateEx(TC_Events.Error.Error1823,FALSE,0);
Error[1824].CreateEx(TC_Events.Error.Error1824,FALSE,0);
Error[1825].CreateEx(TC_Events.Error.Error1825,FALSE,0);
Error[1826].CreateEx(TC_Events.Error.Error1826,FALSE,0);
Error[1827].CreateEx(TC_Events.Error.Error1827,FALSE,0);
Error[1828].CreateEx(TC_Events.Error.Error1828,FALSE,0);
Error[1829].CreateEx(TC_Events.Error.Error1829,FALSE,0);
Error[1830].CreateEx(TC_Events.Error.Error1830,FALSE,0);
Error[1831].CreateEx(TC_Events.Error.Error1831,FALSE,0);
Error[1832].CreateEx(TC_Events.Error.Error1832,FALSE,0);
Error[1833].CreateEx(TC_Events.Error.Error1833,FALSE,0);
Error[1834].CreateEx(TC_Events.Error.Error1834,FALSE,0);
Error[1835].CreateEx(TC_Events.Error.Error1835,FALSE,0);
Error[1836].CreateEx(TC_Events.Error.Error1836,FALSE,0);
Error[1837].CreateEx(TC_Events.Error.Error1837,FALSE,0);
Error[1838].CreateEx(TC_Events.Error.Error1838,FALSE,0);
Error[1839].CreateEx(TC_Events.Error.Error1839,FALSE,0);
Error[1840].CreateEx(TC_Events.Error.Error1840,FALSE,0);
Error[1841].CreateEx(TC_Events.Error.Error1841,FALSE,0);
Error[1842].CreateEx(TC_Events.Error.Error1842,FALSE,0);
Error[1843].CreateEx(TC_Events.Error.Error1843,FALSE,0);
Error[1844].CreateEx(TC_Events.Error.Error1844,FALSE,0);
Error[1845].CreateEx(TC_Events.Error.Error1845,FALSE,0);
Error[1846].CreateEx(TC_Events.Error.Error1846,FALSE,0);
Error[1847].CreateEx(TC_Events.Error.Error1847,FALSE,0);
Error[1848].CreateEx(TC_Events.Error.Error1848,FALSE,0);
Error[1849].CreateEx(TC_Events.Error.Error1849,FALSE,0);
Error[1850].CreateEx(TC_Events.Error.Error1850,FALSE,0);
Error[1851].CreateEx(TC_Events.Error.Error1851,FALSE,0);
Error[1852].CreateEx(TC_Events.Error.Error1852,FALSE,0);
Error[1853].CreateEx(TC_Events.Error.Error1853,FALSE,0);
Error[1854].CreateEx(TC_Events.Error.Error1854,FALSE,0);
Error[1855].CreateEx(TC_Events.Error.Error1855,FALSE,0);
Error[1856].CreateEx(TC_Events.Error.Error1856,FALSE,0);
Error[1857].CreateEx(TC_Events.Error.Error1857,FALSE,0);
Error[1858].CreateEx(TC_Events.Error.Error1858,FALSE,0);
Error[1859].CreateEx(TC_Events.Error.Error1859,FALSE,0);
Error[1860].CreateEx(TC_Events.Error.Error1860,FALSE,0);
Error[1861].CreateEx(TC_Events.Error.Error1861,FALSE,0);
Error[1862].CreateEx(TC_Events.Error.Error1862,FALSE,0);
Error[1863].CreateEx(TC_Events.Error.Error1863,FALSE,0);
Error[1864].CreateEx(TC_Events.Error.Error1864,FALSE,0);
Error[1865].CreateEx(TC_Events.Error.Error1865,FALSE,0);
Error[1866].CreateEx(TC_Events.Error.Error1866,FALSE,0);
Error[1867].CreateEx(TC_Events.Error.Error1867,FALSE,0);
Error[1868].CreateEx(TC_Events.Error.Error1868,FALSE,0);
Error[1869].CreateEx(TC_Events.Error.Error1869,FALSE,0);
Error[1870].CreateEx(TC_Events.Error.Error1870,FALSE,0);
Error[1871].CreateEx(TC_Events.Error.Error1871,FALSE,0);
Error[1872].CreateEx(TC_Events.Error.Error1872,FALSE,0);
Error[1873].CreateEx(TC_Events.Error.Error1873,FALSE,0);
Error[1874].CreateEx(TC_Events.Error.Error1874,FALSE,0);
Error[1875].CreateEx(TC_Events.Error.Error1875,FALSE,0);
Error[1876].CreateEx(TC_Events.Error.Error1876,FALSE,0);
Error[1877].CreateEx(TC_Events.Error.Error1877,FALSE,0);
Error[1878].CreateEx(TC_Events.Error.Error1878,FALSE,0);
Error[1879].CreateEx(TC_Events.Error.Error1879,FALSE,0);
Error[1880].CreateEx(TC_Events.Error.Error1880,FALSE,0);
Error[1881].CreateEx(TC_Events.Error.Error1881,FALSE,0);
Error[1882].CreateEx(TC_Events.Error.Error1882,FALSE,0);
Error[1883].CreateEx(TC_Events.Error.Error1883,FALSE,0);
Error[1884].CreateEx(TC_Events.Error.Error1884,FALSE,0);
Error[1885].CreateEx(TC_Events.Error.Error1885,FALSE,0);
Error[1886].CreateEx(TC_Events.Error.Error1886,FALSE,0);
Error[1887].CreateEx(TC_Events.Error.Error1887,FALSE,0);
Error[1888].CreateEx(TC_Events.Error.Error1888,FALSE,0);
Error[1889].CreateEx(TC_Events.Error.Error1889,FALSE,0);
Error[1890].CreateEx(TC_Events.Error.Error1890,FALSE,0);
Error[1891].CreateEx(TC_Events.Error.Error1891,FALSE,0);
Error[1892].CreateEx(TC_Events.Error.Error1892,FALSE,0);
Error[1893].CreateEx(TC_Events.Error.Error1893,FALSE,0);
Error[1894].CreateEx(TC_Events.Error.Error1894,FALSE,0);
Error[1895].CreateEx(TC_Events.Error.Error1895,FALSE,0);
Error[1896].CreateEx(TC_Events.Error.Error1896,FALSE,0);
Error[1897].CreateEx(TC_Events.Error.Error1897,FALSE,0);
Error[1898].CreateEx(TC_Events.Error.Error1898,FALSE,0);
Error[1899].CreateEx(TC_Events.Error.Error1899,FALSE,0);
Error[1900].CreateEx(TC_Events.Error.Error1900,FALSE,0);
Error[1901].CreateEx(TC_Events.Error.Error1901,FALSE,0);
Error[1902].CreateEx(TC_Events.Error.Error1902,FALSE,0);
Error[1903].CreateEx(TC_Events.Error.Error1903,FALSE,0);
Error[1904].CreateEx(TC_Events.Error.Error1904,FALSE,0);
Error[1905].CreateEx(TC_Events.Error.Error1905,FALSE,0);
Error[1906].CreateEx(TC_Events.Error.Error1906,FALSE,0);
Error[1907].CreateEx(TC_Events.Error.Error1907,FALSE,0);
Error[1908].CreateEx(TC_Events.Error.Error1908,FALSE,0);
Error[1909].CreateEx(TC_Events.Error.Error1909,FALSE,0);
Error[1910].CreateEx(TC_Events.Error.Error1910,FALSE,0);
Error[1911].CreateEx(TC_Events.Error.Error1911,FALSE,0);
Error[1912].CreateEx(TC_Events.Error.Error1912,FALSE,0);
Error[1913].CreateEx(TC_Events.Error.Error1913,FALSE,0);
Error[1914].CreateEx(TC_Events.Error.Error1914,FALSE,0);
Error[1915].CreateEx(TC_Events.Error.Error1915,FALSE,0);
Error[1916].CreateEx(TC_Events.Error.Error1916,FALSE,0);
Error[1917].CreateEx(TC_Events.Error.Error1917,FALSE,0);
Error[1918].CreateEx(TC_Events.Error.Error1918,FALSE,0);
Error[1919].CreateEx(TC_Events.Error.Error1919,FALSE,0);
Error[1920].CreateEx(TC_Events.Error.Error1920,FALSE,0);
Error[1921].CreateEx(TC_Events.Error.Error1921,FALSE,0);
Error[1922].CreateEx(TC_Events.Error.Error1922,FALSE,0);
Error[1923].CreateEx(TC_Events.Error.Error1923,FALSE,0);
Error[1924].CreateEx(TC_Events.Error.Error1924,FALSE,0);
Error[1925].CreateEx(TC_Events.Error.Error1925,FALSE,0);
Error[1926].CreateEx(TC_Events.Error.Error1926,FALSE,0);
Error[1927].CreateEx(TC_Events.Error.Error1927,FALSE,0);
Error[1928].CreateEx(TC_Events.Error.Error1928,FALSE,0);
Error[1929].CreateEx(TC_Events.Error.Error1929,FALSE,0);
Error[1930].CreateEx(TC_Events.Error.Error1930,FALSE,0);
Error[1931].CreateEx(TC_Events.Error.Error1931,FALSE,0);
Error[1932].CreateEx(TC_Events.Error.Error1932,FALSE,0);
Error[1933].CreateEx(TC_Events.Error.Error1933,FALSE,0);
Error[1934].CreateEx(TC_Events.Error.Error1934,FALSE,0);
Error[1935].CreateEx(TC_Events.Error.Error1935,FALSE,0);
Error[1936].CreateEx(TC_Events.Error.Error1936,FALSE,0);
Error[1937].CreateEx(TC_Events.Error.Error1937,FALSE,0);
Error[1938].CreateEx(TC_Events.Error.Error1938,FALSE,0);
Error[1939].CreateEx(TC_Events.Error.Error1939,FALSE,0);
Error[1940].CreateEx(TC_Events.Error.Error1940,FALSE,0);
Error[1941].CreateEx(TC_Events.Error.Error1941,FALSE,0);
Error[1942].CreateEx(TC_Events.Error.Error1942,FALSE,0);
Error[1943].CreateEx(TC_Events.Error.Error1943,FALSE,0);
Error[1944].CreateEx(TC_Events.Error.Error1944,FALSE,0);
Error[1945].CreateEx(TC_Events.Error.Error1945,FALSE,0);
Error[1946].CreateEx(TC_Events.Error.Error1946,FALSE,0);
Error[1947].CreateEx(TC_Events.Error.Error1947,FALSE,0);
Error[1948].CreateEx(TC_Events.Error.Error1948,FALSE,0);
Error[1949].CreateEx(TC_Events.Error.Error1949,FALSE,0);
Error[1950].CreateEx(TC_Events.Error.Error1950,FALSE,0);
Error[1951].CreateEx(TC_Events.Error.Error1951,FALSE,0);
Error[1952].CreateEx(TC_Events.Error.Error1952,FALSE,0);
Error[1953].CreateEx(TC_Events.Error.Error1953,FALSE,0);
Error[1954].CreateEx(TC_Events.Error.Error1954,FALSE,0);
Error[1955].CreateEx(TC_Events.Error.Error1955,FALSE,0);
Error[1956].CreateEx(TC_Events.Error.Error1956,FALSE,0);
Error[1957].CreateEx(TC_Events.Error.Error1957,FALSE,0);
Error[1958].CreateEx(TC_Events.Error.Error1958,FALSE,0);
Error[1959].CreateEx(TC_Events.Error.Error1959,FALSE,0);
Error[1960].CreateEx(TC_Events.Error.Error1960,FALSE,0);
Error[1961].CreateEx(TC_Events.Error.Error1961,FALSE,0);
Error[1962].CreateEx(TC_Events.Error.Error1962,FALSE,0);
Error[1963].CreateEx(TC_Events.Error.Error1963,FALSE,0);
Error[1964].CreateEx(TC_Events.Error.Error1964,FALSE,0);
Error[1965].CreateEx(TC_Events.Error.Error1965,FALSE,0);
Error[1966].CreateEx(TC_Events.Error.Error1966,FALSE,0);
Error[1967].CreateEx(TC_Events.Error.Error1967,FALSE,0);
Error[1968].CreateEx(TC_Events.Error.Error1968,FALSE,0);
Error[1969].CreateEx(TC_Events.Error.Error1969,FALSE,0);
Error[1970].CreateEx(TC_Events.Error.Error1970,FALSE,0);
Error[1971].CreateEx(TC_Events.Error.Error1971,FALSE,0);
Error[1972].CreateEx(TC_Events.Error.Error1972,FALSE,0);
Error[1973].CreateEx(TC_Events.Error.Error1973,FALSE,0);
Error[1974].CreateEx(TC_Events.Error.Error1974,FALSE,0);
Error[1975].CreateEx(TC_Events.Error.Error1975,FALSE,0);
Error[1976].CreateEx(TC_Events.Error.Error1976,FALSE,0);
Error[1977].CreateEx(TC_Events.Error.Error1977,FALSE,0);
Error[1978].CreateEx(TC_Events.Error.Error1978,FALSE,0);
Error[1979].CreateEx(TC_Events.Error.Error1979,FALSE,0);
Error[1980].CreateEx(TC_Events.Error.Error1980,FALSE,0);
Error[1981].CreateEx(TC_Events.Error.Error1981,FALSE,0);
Error[1982].CreateEx(TC_Events.Error.Error1982,FALSE,0);
Error[1983].CreateEx(TC_Events.Error.Error1983,FALSE,0);
Error[1984].CreateEx(TC_Events.Error.Error1984,FALSE,0);
Error[1985].CreateEx(TC_Events.Error.Error1985,FALSE,0);
Error[1986].CreateEx(TC_Events.Error.Error1986,FALSE,0);
Error[1987].CreateEx(TC_Events.Error.Error1987,FALSE,0);
Error[1988].CreateEx(TC_Events.Error.Error1988,FALSE,0);
Error[1989].CreateEx(TC_Events.Error.Error1989,FALSE,0);
Error[1990].CreateEx(TC_Events.Error.Error1990,FALSE,0);
Error[1991].CreateEx(TC_Events.Error.Error1991,FALSE,0);
Error[1992].CreateEx(TC_Events.Error.Error1992,FALSE,0);
Error[1993].CreateEx(TC_Events.Error.Error1993,FALSE,0);
Error[1994].CreateEx(TC_Events.Error.Error1994,FALSE,0);
Error[1995].CreateEx(TC_Events.Error.Error1995,FALSE,0);
Error[1996].CreateEx(TC_Events.Error.Error1996,FALSE,0);
Error[1997].CreateEx(TC_Events.Error.Error1997,FALSE,0);
Error[1998].CreateEx(TC_Events.Error.Error1998,FALSE,0);
Error[1999].CreateEx(TC_Events.Error.Error1999,FALSE,0);
Error[2000].CreateEx(TC_Events.Error.Error2000,FALSE,0);
END_IF
IF NOT bdone THEN
	bdone:=TRUE;
FOR i:=1 TO 2000 BY 1 DO 
	
IF berror[i] THEN
	berror[i]:=FALSE;
	Error[i].Raise(0);
	temp:=TRUE;
END_IF
END_FOR
bdone:=FALSE;
END_IF

IF reset THEN
	FOR j:=1 TO 2000 BY 1 DO 
	bclear[j]:=FALSE;
	Error[j].Clear(0,TRUE);
	END_FOR
	temp:=false;
END_IF

berror[1]:=Bin1;
berror[2]:=Bin2;
berror[3]:=Bin3;
berror[4]:=Bin4;
berror[101]:=Bin5;
berror[102]:=Bin6;
berror[103]:=Bin7;

(*IF bInit THEN
	bInit:=FALSE;
	Error[1].CreateEx(TC_Events.Error.Error1,TRUE,0);
END_IF

IF bRaise THEN
	bRaise:=FALSE;
	Error[1].Raise(0);
END_IF

IF bclearA THEN
	bclearA := FALSE;
	Error[1].Clear(0,TRUE);
END_IF;*)

END_PROGRAM

// ---- POUs/Programs/OP10/OP10_ROBO.TcPOU
PROGRAM OP10_ROBO
VAR
	I_OP10A_6000_6007						: BYTE_AS_BIT;	
	I_OP10A_6008_6015                       : BYTE_AS_BIT;
	I_OP10A_6016_6023                       : BYTE_AS_BIT;
	I_OP10A_6024_6031                       : BYTE_AS_BIT;
	I_OP10A_6032_6039                       : BYTE_AS_BIT;
	I_OP10A_6040_6047                       : BYTE_AS_BIT;
	I_OP10A_6048_6055                       : BYTE_AS_BIT;
	I_OP10A_6056_6063                       : BYTE_AS_BIT;
	O_OP10A_6000_6007						: BIT_AS_BYTE;
	O_OP10A_6008_6015						: BIT_AS_BYTE;
	O_OP10A_6016_6023						: BIT_AS_BYTE;
	O_OP10A_6024_6031						: BIT_AS_BYTE;
	O_OP10A_6032_6039						: BIT_AS_BYTE;
	O_OP10A_6040_6047						: BIT_AS_BYTE;
	O_OP10A_6048_6055						: BIT_AS_BYTE;
	O_OP10A_6056_6063						: BIT_AS_BYTE;

	I_OP10B_6000_6007						: BYTE_AS_BIT;	
	I_OP10B_6008_6015                       : BYTE_AS_BIT;
	I_OP10B_6016_6023                       : BYTE_AS_BIT;
	I_OP10B_6024_6031                       : BYTE_AS_BIT;
	I_OP10B_6032_6039                       : BYTE_AS_BIT;
	I_OP10B_6040_6047                       : BYTE_AS_BIT;
	I_OP10B_6048_6055                       : BYTE_AS_BIT;
	I_OP10B_6056_6063                       : BYTE_AS_BIT;
	O_OP10B_6032_6039						: BIT_AS_BYTE;
	O_OP10B_6040_6047						: BIT_AS_BYTE;
	O_OP10B_6048_6055						: BIT_AS_BYTE;
	O_OP10B_6056_6063						: BIT_AS_BYTE;
	O_OP10B_6000_6007						: BIT_AS_BYTE;
	O_OP10B_6008_6015						: BIT_AS_BYTE;
	O_OP10B_6016_6023						: BIT_AS_BYTE;
	O_OP10B_6024_6031						: BIT_AS_BYTE;

	OP10A_IP_ROBO_6000_6007  AT %I*			: USINT;
	OP10A_IP_ROBO_6008_6015  AT %I*			: USINT;
	OP10A_IP_ROBO_6016_6023  AT %I*			: USINT;
	OP10A_IP_ROBO_6024_6031  AT %I*			: USINT;
	OP10A_IP_ROBO_6032_6039  AT %I*			: USINT;
	OP10A_IP_ROBO_6040_6047  AT %I*			: USINT;	
	OP10A_IP_ROBO_6048_6055  AT %I*			: USINT;	
	OP10A_IP_ROBO_6056_6063  AT %I*			: USINT;	
	OP10A_OP_ROBO_6000_6007  AT %Q*			: USINT;
	OP10A_OP_ROBO_6008_6015  AT %Q*			: USINT;
	OP10A_OP_ROBO_6016_6023  AT %Q*			: USINT;
	OP10A_OP_ROBO_6024_6031  AT %Q*			: USINT;
	OP10A_OP_ROBO_6032_6039  AT %Q*			: USINT;
	OP10A_OP_ROBO_6040_6047  AT %Q*			: USINT;	
	OP10A_OP_ROBO_6048_6055  AT %Q*			: USINT;	
	OP10A_OP_ROBO_6056_6063  AT %Q*			: USINT;

	OP10B_IP_ROBO_6000_6007  AT %I*			: USINT;
	OP10B_IP_ROBO_6008_6015  AT %I*			: USINT;
	OP10B_IP_ROBO_6016_6023  AT %I*			: USINT;
	OP10B_IP_ROBO_6024_6031  AT %I*			: USINT;
	OP10B_IP_ROBO_6032_6039  AT %I*			: USINT;
	OP10B_IP_ROBO_6040_6047  AT %I*			: USINT;	
	OP10B_IP_ROBO_6048_6055  AT %I*			: USINT;	
	OP10B_IP_ROBO_6056_6063  AT %I*			: USINT;
	OP10B_OP_ROBO_6000_6007  AT %Q*			: USINT;
	OP10B_OP_ROBO_6008_6015  AT %Q*			: USINT;
	OP10B_OP_ROBO_6016_6023  AT %Q*			: USINT;
	OP10B_OP_ROBO_6024_6031  AT %Q*			: USINT;
	OP10B_OP_ROBO_6032_6039  AT %Q*			: USINT;
	OP10B_OP_ROBO_6040_6047  AT %Q*			: USINT;	
	OP10B_OP_ROBO_6048_6055  AT %Q*			: USINT;	
	OP10B_OP_ROBO_6056_6063  AT %Q*			: USINT;	


	


END_VAR

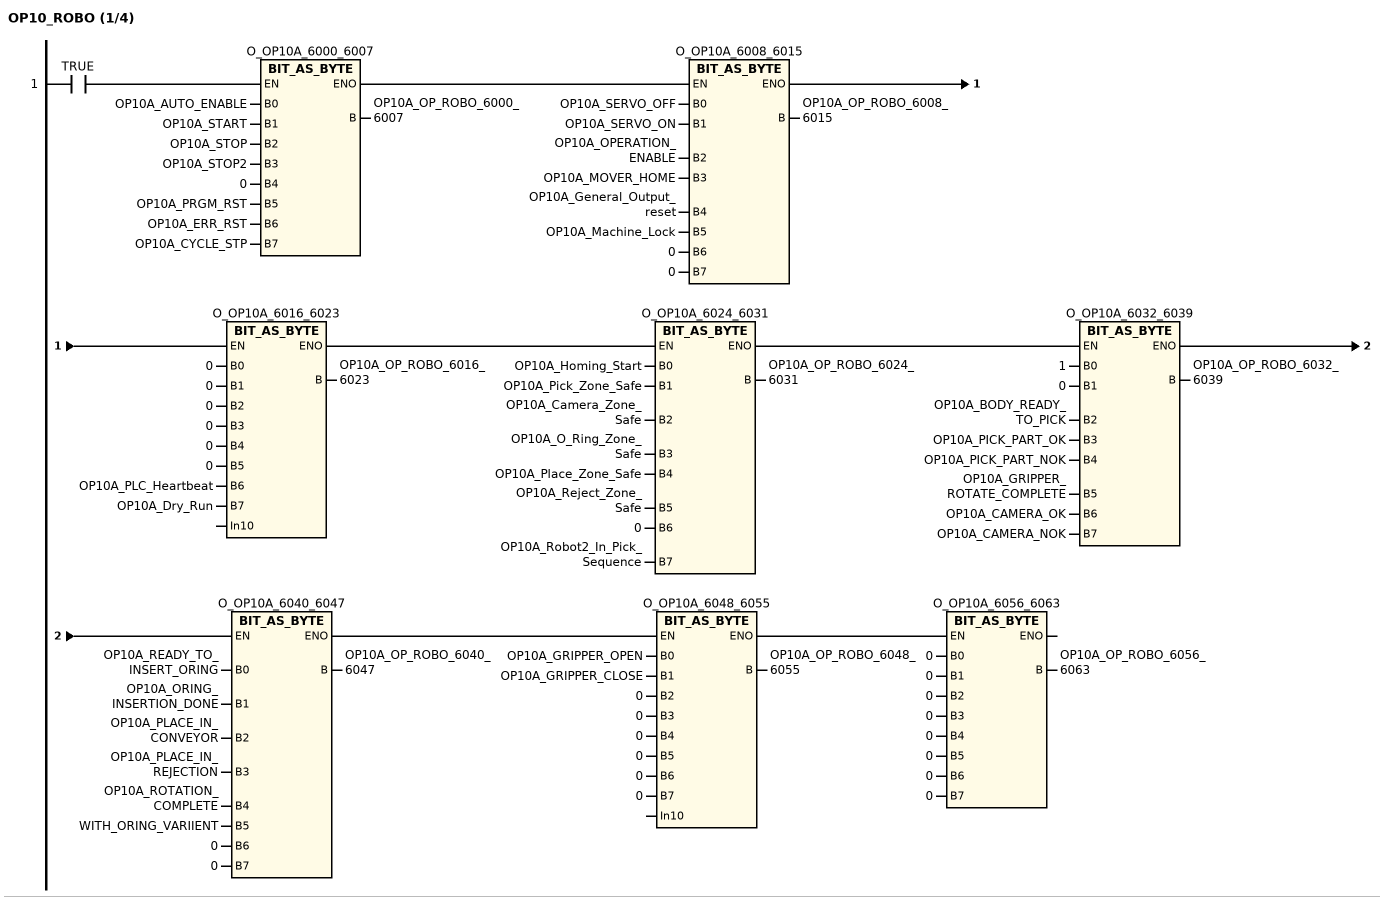
// NETWORK 1
O_OP10A_6000_6007(
    B0 := OP10A_AUTO_ENABLE,
    B1 := OP10A_START,
    B2 := OP10A_STOP,
    B3 := OP10A_STOP2,
    B4 := 0,
    B5 := OP10A_PRGM_RST,
    B6 := OP10A_ERR_RST,
    B7 := OP10A_CYCLE_STP,
    B => OP10A_OP_ROBO_6000_6007); // BIT_AS_BYTE
O_OP10A_6008_6015(
    B0 := OP10A_SERVO_OFF,
    B1 := OP10A_SERVO_ON,
    B2 := OP10A_OPERATION_ENABLE,
    B3 := OP10A_MOVER_HOME,
    B4 := OP10A_General_Output_reset,
    B5 := OP10A_Machine_Lock,
    B6 := 0,
    B7 := 0,
    B => OP10A_OP_ROBO_6008_6015); // BIT_AS_BYTE
O_OP10A_6016_6023(
    B0 := 0,
    B1 := 0,
    B2 := 0,
    B3 := 0,
    B4 := 0,
    B5 := 0,
    B6 := OP10A_PLC_Heartbeat,
    B7 := OP10A_Dry_Run,
    B => OP10A_OP_ROBO_6016_6023); // BIT_AS_BYTE
O_OP10A_6024_6031(
    B0 := OP10A_Homing_Start,
    B1 := OP10A_Pick_Zone_Safe,
    B2 := OP10A_Camera_Zone_Safe,
    B3 := OP10A_O_Ring_Zone_Safe,
    B4 := OP10A_Place_Zone_Safe,
    B5 := OP10A_Reject_Zone_Safe,
    B6 := 0,
    B7 := OP10A_Robot2_In_Pick_Sequence,
    B => OP10A_OP_ROBO_6024_6031); // BIT_AS_BYTE
O_OP10A_6032_6039(
    B0 := 1,
    B1 := 0,
    B2 := OP10A_BODY_READY_TO_PICK,
    B3 := OP10A_PICK_PART_OK,
    B4 := OP10A_PICK_PART_NOK,
    B5 := OP10A_GRIPPER_ROTATE_COMPLETE,
    B6 := OP10A_CAMERA_OK,
    B7 := OP10A_CAMERA_NOK,
    B => OP10A_OP_ROBO_6032_6039); // BIT_AS_BYTE
O_OP10A_6040_6047(
    B0 := OP10A_READY_TO_INSERT_ORING,
    B1 := OP10A_ORING_INSERTION_DONE,
    B2 := OP10A_PLACE_IN_CONVEYOR,
    B3 := OP10A_PLACE_IN_REJECTION,
    B4 := OP10A_ROTATION_COMPLETE,
    B5 := WITH_ORING_VARIIENT,
    B6 := 0,
    B7 := 0,
    B => OP10A_OP_ROBO_6040_6047); // BIT_AS_BYTE
O_OP10A_6048_6055(
    B0 := OP10A_GRIPPER_OPEN,
    B1 := OP10A_GRIPPER_CLOSE,
    B2 := 0,
    B3 := 0,
    B4 := 0,
    B5 := 0,
    B6 := 0,
    B7 := 0,
    B => OP10A_OP_ROBO_6048_6055); // BIT_AS_BYTE
O_OP10A_6056_6063(
    B0 := 0,
    B1 := 0,
    B2 := 0,
    B3 := 0,
    B4 := 0,
    B5 := 0,
    B6 := 0,
    B7 := 0,
    B => OP10A_OP_ROBO_6056_6063); // BIT_AS_BYTE

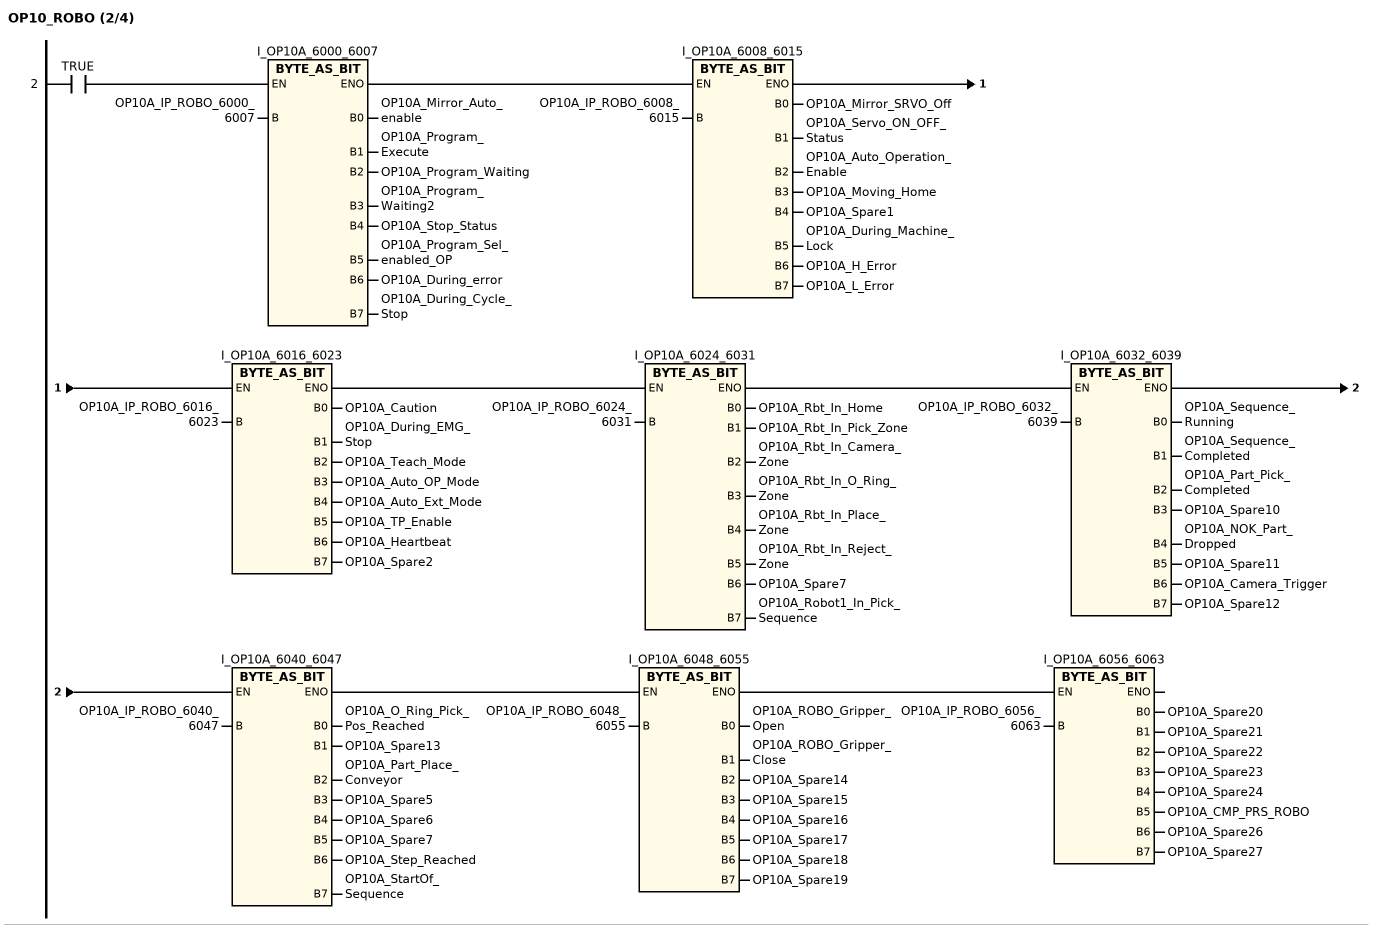
// NETWORK 2
I_OP10A_6000_6007(
    B := OP10A_IP_ROBO_6000_6007,
    B0 => OP10A_Mirror_Auto_enable,
    B1 => OP10A_Program_Execute,
    B2 => OP10A_Program_Waiting,
    B3 => OP10A_Program_Waiting2,
    B4 => OP10A_Stop_Status,
    B5 => OP10A_Program_Sel_enabled_OP,
    B6 => OP10A_During_error,
    B7 => OP10A_During_Cycle_Stop); // BYTE_AS_BIT
I_OP10A_6008_6015(
    B := OP10A_IP_ROBO_6008_6015,
    B0 => OP10A_Mirror_SRVO_Off,
    B1 => OP10A_Servo_ON_OFF_Status,
    B2 => OP10A_Auto_Operation_Enable,
    B3 => OP10A_Moving_Home,
    B4 => OP10A_Spare1,
    B5 => OP10A_During_Machine_Lock,
    B6 => OP10A_H_Error,
    B7 => OP10A_L_Error); // BYTE_AS_BIT
I_OP10A_6016_6023(
    B := OP10A_IP_ROBO_6016_6023,
    B0 => OP10A_Caution,
    B1 => OP10A_During_EMG_Stop,
    B2 => OP10A_Teach_Mode,
    B3 => OP10A_Auto_OP_Mode,
    B4 => OP10A_Auto_Ext_Mode,
    B5 => OP10A_TP_Enable,
    B6 => OP10A_Heartbeat,
    B7 => OP10A_Spare2); // BYTE_AS_BIT
I_OP10A_6024_6031(
    B := OP10A_IP_ROBO_6024_6031,
    B0 => OP10A_Rbt_In_Home,
    B1 => OP10A_Rbt_In_Pick_Zone,
    B2 => OP10A_Rbt_In_Camera_Zone,
    B3 => OP10A_Rbt_In_O_Ring_Zone,
    B4 => OP10A_Rbt_In_Place_Zone,
    B5 => OP10A_Rbt_In_Reject_Zone,
    B6 => OP10A_Spare7,
    B7 => OP10A_Robot1_In_Pick_Sequence); // BYTE_AS_BIT
I_OP10A_6032_6039(
    B := OP10A_IP_ROBO_6032_6039,
    B0 => OP10A_Sequence_Running,
    B1 => OP10A_Sequence_Completed,
    B2 => OP10A_Part_Pick_Completed,
    B3 => OP10A_Spare10,
    B4 => OP10A_NOK_Part_Dropped,
    B5 => OP10A_Spare11,
    B6 => OP10A_Camera_Trigger,
    B7 => OP10A_Spare12); // BYTE_AS_BIT
I_OP10A_6040_6047(
    B := OP10A_IP_ROBO_6040_6047,
    B0 => OP10A_O_Ring_Pick_Pos_Reached,
    B1 => OP10A_Spare13,
    B2 => OP10A_Part_Place_Conveyor,
    B3 => OP10A_Spare5,
    B4 => OP10A_Spare6,
    B5 => OP10A_Spare7,
    B6 => OP10A_Step_Reached,
    B7 => OP10A_StartOf_Sequence); // BYTE_AS_BIT
I_OP10A_6048_6055(
    B := OP10A_IP_ROBO_6048_6055,
    B0 => OP10A_ROBO_Gripper_Open,
    B1 => OP10A_ROBO_Gripper_Close,
    B2 => OP10A_Spare14,
    B3 => OP10A_Spare15,
    B4 => OP10A_Spare16,
    B5 => OP10A_Spare17,
    B6 => OP10A_Spare18,
    B7 => OP10A_Spare19); // BYTE_AS_BIT
I_OP10A_6056_6063(
    B := OP10A_IP_ROBO_6056_6063,
    B0 => OP10A_Spare20,
    B1 => OP10A_Spare21,
    B2 => OP10A_Spare22,
    B3 => OP10A_Spare23,
    B4 => OP10A_Spare24,
    B5 => OP10A_CMP_PRS_ROBO,
    B6 => OP10A_Spare26,
    B7 => OP10A_Spare27); // BYTE_AS_BIT

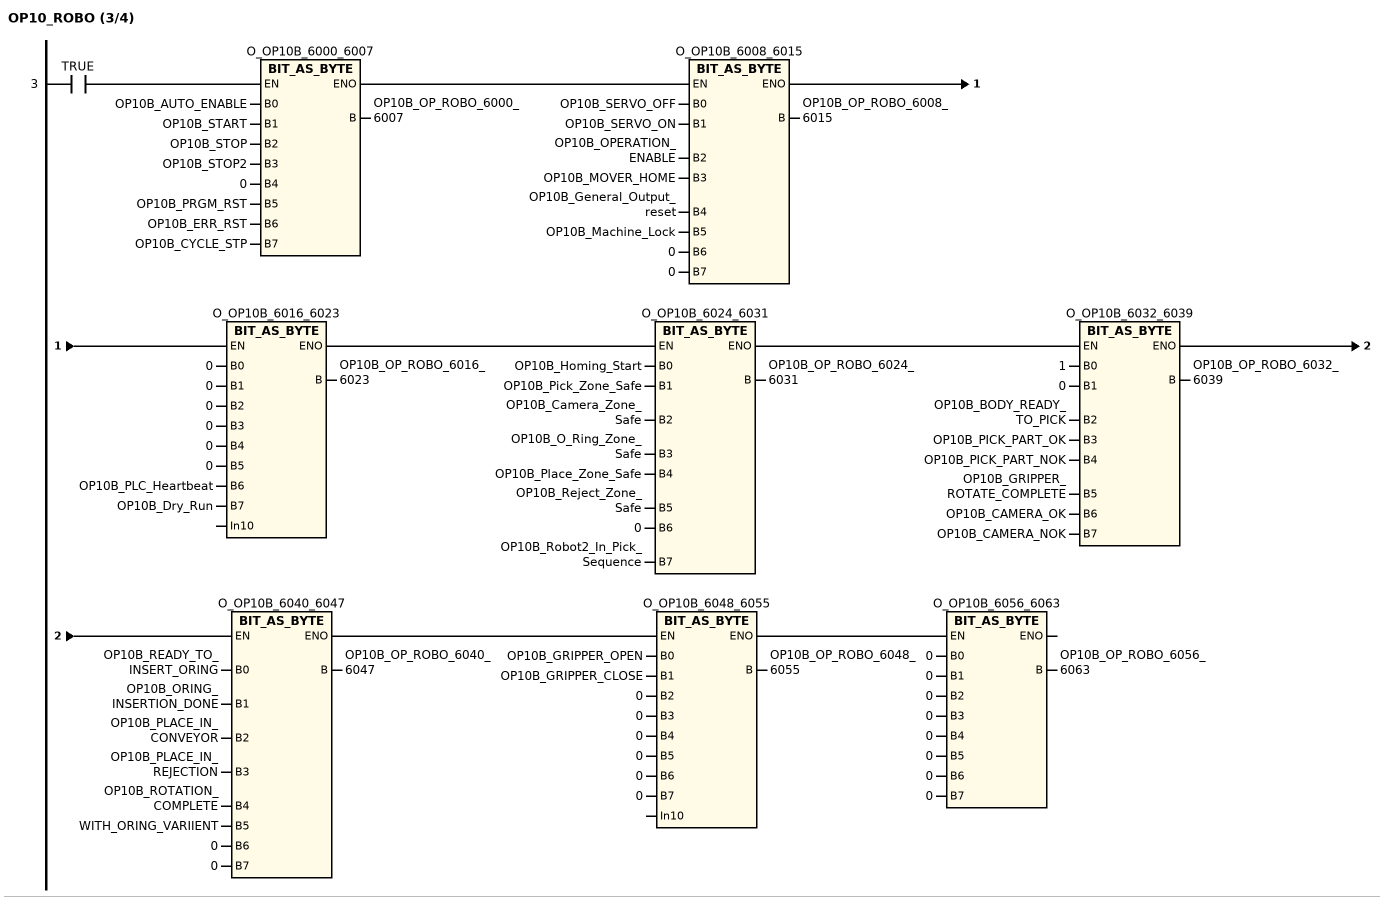
// NETWORK 3
O_OP10B_6000_6007(
    B0 := OP10B_AUTO_ENABLE,
    B1 := OP10B_START,
    B2 := OP10B_STOP,
    B3 := OP10B_STOP2,
    B4 := 0,
    B5 := OP10B_PRGM_RST,
    B6 := OP10B_ERR_RST,
    B7 := OP10B_CYCLE_STP,
    B => OP10B_OP_ROBO_6000_6007); // BIT_AS_BYTE
O_OP10B_6008_6015(
    B0 := OP10B_SERVO_OFF,
    B1 := OP10B_SERVO_ON,
    B2 := OP10B_OPERATION_ENABLE,
    B3 := OP10B_MOVER_HOME,
    B4 := OP10B_General_Output_reset,
    B5 := OP10B_Machine_Lock,
    B6 := 0,
    B7 := 0,
    B => OP10B_OP_ROBO_6008_6015); // BIT_AS_BYTE
O_OP10B_6016_6023(
    B0 := 0,
    B1 := 0,
    B2 := 0,
    B3 := 0,
    B4 := 0,
    B5 := 0,
    B6 := OP10B_PLC_Heartbeat,
    B7 := OP10B_Dry_Run,
    B => OP10B_OP_ROBO_6016_6023); // BIT_AS_BYTE
O_OP10B_6024_6031(
    B0 := OP10B_Homing_Start,
    B1 := OP10B_Pick_Zone_Safe,
    B2 := OP10B_Camera_Zone_Safe,
    B3 := OP10B_O_Ring_Zone_Safe,
    B4 := OP10B_Place_Zone_Safe,
    B5 := OP10B_Reject_Zone_Safe,
    B6 := 0,
    B7 := OP10B_Robot2_In_Pick_Sequence,
    B => OP10B_OP_ROBO_6024_6031); // BIT_AS_BYTE
O_OP10B_6032_6039(
    B0 := 1,
    B1 := 0,
    B2 := OP10B_BODY_READY_TO_PICK,
    B3 := OP10B_PICK_PART_OK,
    B4 := OP10B_PICK_PART_NOK,
    B5 := OP10B_GRIPPER_ROTATE_COMPLETE,
    B6 := OP10B_CAMERA_OK,
    B7 := OP10B_CAMERA_NOK,
    B => OP10B_OP_ROBO_6032_6039); // BIT_AS_BYTE
O_OP10B_6040_6047(
    B0 := OP10B_READY_TO_INSERT_ORING,
    B1 := OP10B_ORING_INSERTION_DONE,
    B2 := OP10B_PLACE_IN_CONVEYOR,
    B3 := OP10B_PLACE_IN_REJECTION,
    B4 := OP10B_ROTATION_COMPLETE,
    B5 := WITH_ORING_VARIIENT,
    B6 := 0,
    B7 := 0,
    B => OP10B_OP_ROBO_6040_6047); // BIT_AS_BYTE
O_OP10B_6048_6055(
    B0 := OP10B_GRIPPER_OPEN,
    B1 := OP10B_GRIPPER_CLOSE,
    B2 := 0,
    B3 := 0,
    B4 := 0,
    B5 := 0,
    B6 := 0,
    B7 := 0,
    B => OP10B_OP_ROBO_6048_6055); // BIT_AS_BYTE
O_OP10B_6056_6063(
    B0 := 0,
    B1 := 0,
    B2 := 0,
    B3 := 0,
    B4 := 0,
    B5 := 0,
    B6 := 0,
    B7 := 0,
    B => OP10B_OP_ROBO_6056_6063); // BIT_AS_BYTE

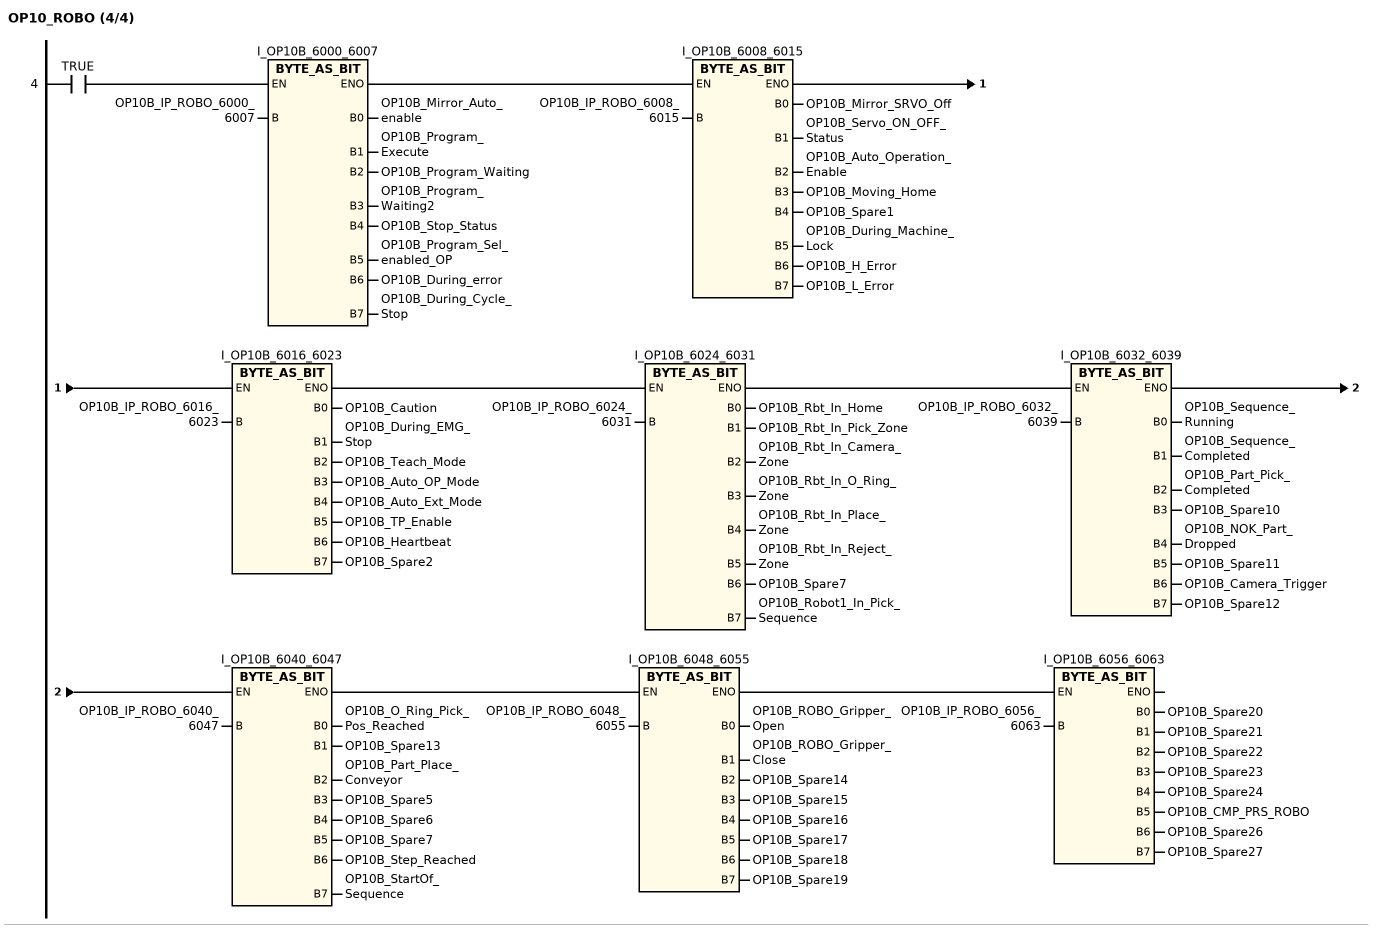
// NETWORK 4
I_OP10B_6000_6007(
    B := OP10B_IP_ROBO_6000_6007,
    B0 => OP10B_Mirror_Auto_enable,
    B1 => OP10B_Program_Execute,
    B2 => OP10B_Program_Waiting,
    B3 => OP10B_Program_Waiting2,
    B4 => OP10B_Stop_Status,
    B5 => OP10B_Program_Sel_enabled_OP,
    B6 => OP10B_During_error,
    B7 => OP10B_During_Cycle_Stop); // BYTE_AS_BIT
I_OP10B_6008_6015(
    B := OP10B_IP_ROBO_6008_6015,
    B0 => OP10B_Mirror_SRVO_Off,
    B1 => OP10B_Servo_ON_OFF_Status,
    B2 => OP10B_Auto_Operation_Enable,
    B3 => OP10B_Moving_Home,
    B4 => OP10B_Spare1,
    B5 => OP10B_During_Machine_Lock,
    B6 => OP10B_H_Error,
    B7 => OP10B_L_Error); // BYTE_AS_BIT
I_OP10B_6016_6023(
    B := OP10B_IP_ROBO_6016_6023,
    B0 => OP10B_Caution,
    B1 => OP10B_During_EMG_Stop,
    B2 => OP10B_Teach_Mode,
    B3 => OP10B_Auto_OP_Mode,
    B4 => OP10B_Auto_Ext_Mode,
    B5 => OP10B_TP_Enable,
    B6 => OP10B_Heartbeat,
    B7 => OP10B_Spare2); // BYTE_AS_BIT
I_OP10B_6024_6031(
    B := OP10B_IP_ROBO_6024_6031,
    B0 => OP10B_Rbt_In_Home,
    B1 => OP10B_Rbt_In_Pick_Zone,
    B2 => OP10B_Rbt_In_Camera_Zone,
    B3 => OP10B_Rbt_In_O_Ring_Zone,
    B4 => OP10B_Rbt_In_Place_Zone,
    B5 => OP10B_Rbt_In_Reject_Zone,
    B6 => OP10B_Spare7,
    B7 => OP10B_Robot1_In_Pick_Sequence); // BYTE_AS_BIT
I_OP10B_6032_6039(
    B := OP10B_IP_ROBO_6032_6039,
    B0 => OP10B_Sequence_Running,
    B1 => OP10B_Sequence_Completed,
    B2 => OP10B_Part_Pick_Completed,
    B3 => OP10B_Spare10,
    B4 => OP10B_NOK_Part_Dropped,
    B5 => OP10B_Spare11,
    B6 => OP10B_Camera_Trigger,
    B7 => OP10B_Spare12); // BYTE_AS_BIT
I_OP10B_6040_6047(
    B := OP10B_IP_ROBO_6040_6047,
    B0 => OP10B_O_Ring_Pick_Pos_Reached,
    B1 => OP10B_Spare13,
    B2 => OP10B_Part_Place_Conveyor,
    B3 => OP10B_Spare5,
    B4 => OP10B_Spare6,
    B5 => OP10B_Spare7,
    B6 => OP10B_Step_Reached,
    B7 => OP10B_StartOf_Sequence); // BYTE_AS_BIT
I_OP10B_6048_6055(
    B := OP10B_IP_ROBO_6048_6055,
    B0 => OP10B_ROBO_Gripper_Open,
    B1 => OP10B_ROBO_Gripper_Close,
    B2 => OP10B_Spare14,
    B3 => OP10B_Spare15,
    B4 => OP10B_Spare16,
    B5 => OP10B_Spare17,
    B6 => OP10B_Spare18,
    B7 => OP10B_Spare19); // BYTE_AS_BIT
I_OP10B_6056_6063(
    B := OP10B_IP_ROBO_6056_6063,
    B0 => OP10B_Spare20,
    B1 => OP10B_Spare21,
    B2 => OP10B_Spare22,
    B3 => OP10B_Spare23,
    B4 => OP10B_Spare24,
    B5 => OP10B_CMP_PRS_ROBO,
    B6 => OP10B_Spare26,
    B7 => OP10B_Spare27); // BYTE_AS_BIT

END_PROGRAM

// ---- POUs/Programs/OP160/OP160_Robo_Byte_Mapping.TcPOU
PROGRAM OP160_Robo_Byte_Mapping
VAR

//registerout

	OP160_Robo_IN_Byte2: BYTE_AS_BIT;
	OP160_Robo_IN_Byte3: BYTE_AS_BIT;
	OP160_Robo_IN_Byte4: BYTE_AS_BIT;
	OP160_Robo_IN_Byte5: BYTE_AS_BIT;
	OP160_Robo_IN_Byte6: BYTE_AS_BIT;
	OP160_Robo_IN_Byte7: BYTE_AS_BIT;
	OP160_Robo_IN_Byte8: BYTE_AS_BIT;
	OP160_Robo_Out_Byte1: BIT_AS_BYTE;
	OP160_Robo_Out_Byte2: BIT_AS_BYTE;
	OP160_Robo_Out_Byte3: BIT_AS_BYTE;
	OP160_Robo_Out_Byte4: BIT_AS_BYTE;
	OP160_Robo_Out_Byte5: BIT_AS_BYTE;
	OP160_Robo_Out_Byte6: BIT_AS_BYTE;
	OP160_Robo_Out_Byte7: BIT_AS_BYTE;
	OP160_Robo_Out_Byte8: BIT_AS_BYTE;
	OP160_EI_Rdy_Reject: BOOL;
END_VAR

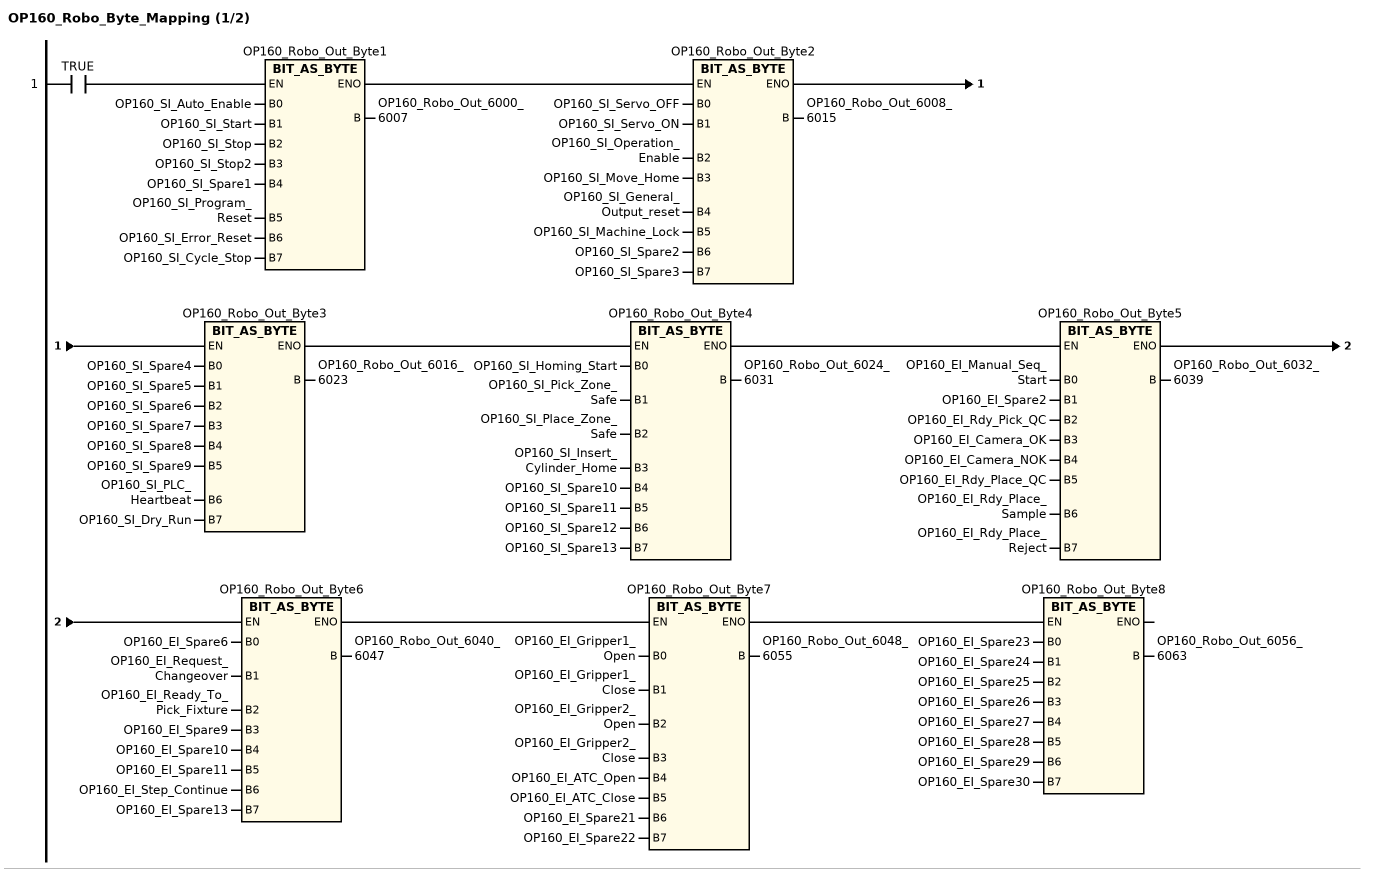
// NETWORK 1
OP160_Robo_Out_Byte1(
    B0 := OP160_SI_Auto_Enable,
    B1 := OP160_SI_Start,
    B2 := OP160_SI_Stop,
    B3 := OP160_SI_Stop2,
    B4 := OP160_SI_Spare1,
    B5 := OP160_SI_Program_Reset,
    B6 := OP160_SI_Error_Reset,
    B7 := OP160_SI_Cycle_Stop,
    B => OP160_Robo_Out_6000_6007); // BIT_AS_BYTE
OP160_Robo_Out_Byte2(
    B0 := OP160_SI_Servo_OFF,
    B1 := OP160_SI_Servo_ON,
    B2 := OP160_SI_Operation_Enable,
    B3 := OP160_SI_Move_Home,
    B4 := OP160_SI_General_Output_reset,
    B5 := OP160_SI_Machine_Lock,
    B6 := OP160_SI_Spare2,
    B7 := OP160_SI_Spare3,
    B => OP160_Robo_Out_6008_6015); // BIT_AS_BYTE
OP160_Robo_Out_Byte3(
    B0 := OP160_SI_Spare4,
    B1 := OP160_SI_Spare5,
    B2 := OP160_SI_Spare6,
    B3 := OP160_SI_Spare7,
    B4 := OP160_SI_Spare8,
    B5 := OP160_SI_Spare9,
    B6 := OP160_SI_PLC_Heartbeat,
    B7 := OP160_SI_Dry_Run,
    B => OP160_Robo_Out_6016_6023); // BIT_AS_BYTE
OP160_Robo_Out_Byte4(
    B0 := OP160_SI_Homing_Start,
    B1 := OP160_SI_Pick_Zone_Safe,
    B2 := OP160_SI_Place_Zone_Safe,
    B3 := OP160_SI_Insert_Cylinder_Home,
    B4 := OP160_SI_Spare10,
    B5 := OP160_SI_Spare11,
    B6 := OP160_SI_Spare12,
    B7 := OP160_SI_Spare13,
    B => OP160_Robo_Out_6024_6031); // BIT_AS_BYTE
OP160_Robo_Out_Byte5(
    B0 := OP160_EI_Manual_Seq_Start,
    B1 := OP160_EI_Spare2,
    B2 := OP160_EI_Rdy_Pick_QC,
    B3 := OP160_EI_Camera_OK,
    B4 := OP160_EI_Camera_NOK,
    B5 := OP160_EI_Rdy_Place_QC,
    B6 := OP160_EI_Rdy_Place_Sample,
    B7 := OP160_EI_Rdy_Place_Reject,
    B => OP160_Robo_Out_6032_6039); // BIT_AS_BYTE
OP160_Robo_Out_Byte6(
    B0 := OP160_EI_Spare6,
    B1 := OP160_EI_Request_Changeover,
    B2 := OP160_EI_Ready_To_Pick_Fixture,
    B3 := OP160_EI_Spare9,
    B4 := OP160_EI_Spare10,
    B5 := OP160_EI_Spare11,
    B6 := OP160_EI_Step_Continue,
    B7 := OP160_EI_Spare13,
    B => OP160_Robo_Out_6040_6047); // BIT_AS_BYTE
OP160_Robo_Out_Byte7(
    B0 := OP160_EI_Gripper1_Open,
    B1 := OP160_EI_Gripper1_Close,
    B2 := OP160_EI_Gripper2_Open,
    B3 := OP160_EI_Gripper2_Close,
    B4 := OP160_EI_ATC_Open,
    B5 := OP160_EI_ATC_Close,
    B6 := OP160_EI_Spare21,
    B7 := OP160_EI_Spare22,
    B => OP160_Robo_Out_6048_6055); // BIT_AS_BYTE
OP160_Robo_Out_Byte8(
    B0 := OP160_EI_Spare23,
    B1 := OP160_EI_Spare24,
    B2 := OP160_EI_Spare25,
    B3 := OP160_EI_Spare26,
    B4 := OP160_EI_Spare27,
    B5 := OP160_EI_Spare28,
    B6 := OP160_EI_Spare29,
    B7 := OP160_EI_Spare30,
    B => OP160_Robo_Out_6056_6063); // BIT_AS_BYTE

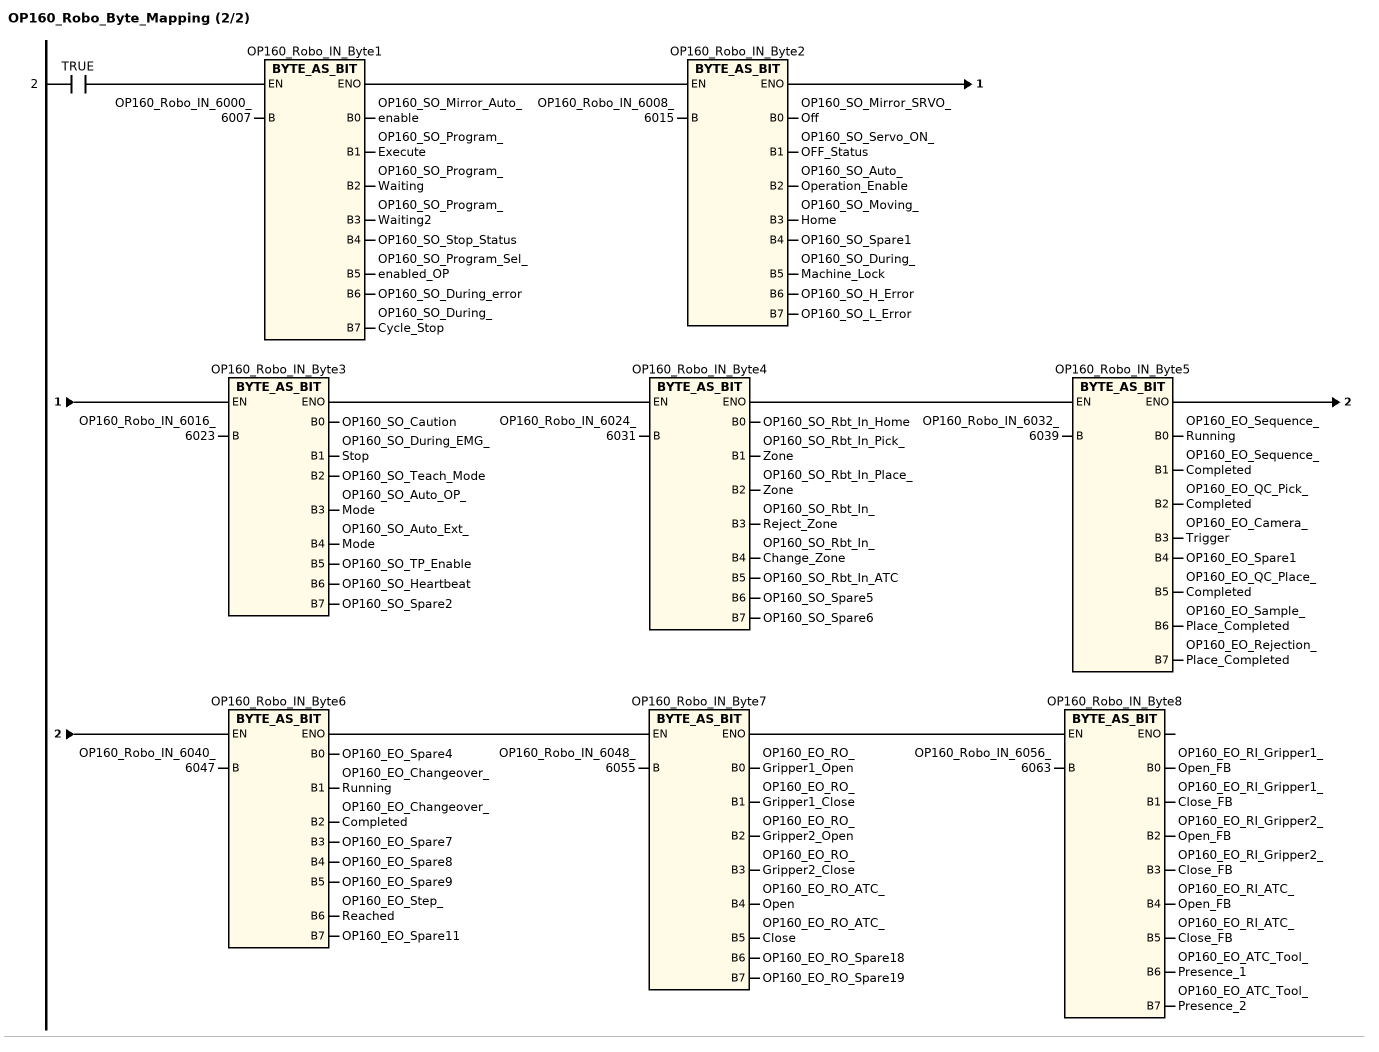
// NETWORK 2
OP160_Robo_IN_Byte1(
    B := OP160_Robo_IN_6000_6007,
    B0 => OP160_SO_Mirror_Auto_enable,
    B1 => OP160_SO_Program_Execute,
    B2 => OP160_SO_Program_Waiting,
    B3 => OP160_SO_Program_Waiting2,
    B4 => OP160_SO_Stop_Status,
    B5 => OP160_SO_Program_Sel_enabled_OP,
    B6 => OP160_SO_During_error,
    B7 => OP160_SO_During_Cycle_Stop); // BYTE_AS_BIT
OP160_Robo_IN_Byte2(
    B := OP160_Robo_IN_6008_6015,
    B0 => OP160_SO_Mirror_SRVO_Off,
    B1 => OP160_SO_Servo_ON_OFF_Status,
    B2 => OP160_SO_Auto_Operation_Enable,
    B3 => OP160_SO_Moving_Home,
    B4 => OP160_SO_Spare1,
    B5 => OP160_SO_During_Machine_Lock,
    B6 => OP160_SO_H_Error,
    B7 => OP160_SO_L_Error); // BYTE_AS_BIT
OP160_Robo_IN_Byte3(
    B := OP160_Robo_IN_6016_6023,
    B0 => OP160_SO_Caution,
    B1 => OP160_SO_During_EMG_Stop,
    B2 => OP160_SO_Teach_Mode,
    B3 => OP160_SO_Auto_OP_Mode,
    B4 => OP160_SO_Auto_Ext_Mode,
    B5 => OP160_SO_TP_Enable,
    B6 => OP160_SO_Heartbeat,
    B7 => OP160_SO_Spare2); // BYTE_AS_BIT
OP160_Robo_IN_Byte4(
    B := OP160_Robo_IN_6024_6031,
    B0 => OP160_SO_Rbt_In_Home,
    B1 => OP160_SO_Rbt_In_Pick_Zone,
    B2 => OP160_SO_Rbt_In_Place_Zone,
    B3 => OP160_SO_Rbt_In_Reject_Zone,
    B4 => OP160_SO_Rbt_In_Change_Zone,
    B5 => OP160_SO_Rbt_In_ATC,
    B6 => OP160_SO_Spare5,
    B7 => OP160_SO_Spare6); // BYTE_AS_BIT
OP160_Robo_IN_Byte5(
    B := OP160_Robo_IN_6032_6039,
    B0 => OP160_EO_Sequence_Running,
    B1 => OP160_EO_Sequence_Completed,
    B2 => OP160_EO_QC_Pick_Completed,
    B3 => OP160_EO_Camera_Trigger,
    B4 => OP160_EO_Spare1,
    B5 => OP160_EO_QC_Place_Completed,
    B6 => OP160_EO_Sample_Place_Completed,
    B7 => OP160_EO_Rejection_Place_Completed); // BYTE_AS_BIT
OP160_Robo_IN_Byte6(
    B := OP160_Robo_IN_6040_6047,
    B0 => OP160_EO_Spare4,
    B1 => OP160_EO_Changeover_Running,
    B2 => OP160_EO_Changeover_Completed,
    B3 => OP160_EO_Spare7,
    B4 => OP160_EO_Spare8,
    B5 => OP160_EO_Spare9,
    B6 => OP160_EO_Step_Reached,
    B7 => OP160_EO_Spare11); // BYTE_AS_BIT
OP160_Robo_IN_Byte7(
    B := OP160_Robo_IN_6048_6055,
    B0 => OP160_EO_RO_Gripper1_Open,
    B1 => OP160_EO_RO_Gripper1_Close,
    B2 => OP160_EO_RO_Gripper2_Open,
    B3 => OP160_EO_RO_Gripper2_Close,
    B4 => OP160_EO_RO_ATC_Open,
    B5 => OP160_EO_RO_ATC_Close,
    B6 => OP160_EO_RO_Spare18,
    B7 => OP160_EO_RO_Spare19); // BYTE_AS_BIT
OP160_Robo_IN_Byte8(
    B := OP160_Robo_IN_6056_6063,
    B0 => OP160_EO_RI_Gripper1_Open_FB,
    B1 => OP160_EO_RI_Gripper1_Close_FB,
    B2 => OP160_EO_RI_Gripper2_Open_FB,
    B3 => OP160_EO_RI_Gripper2_Close_FB,
    B4 => OP160_EO_RI_ATC_Open_FB,
    B5 => OP160_EO_RI_ATC_Close_FB,
    B6 => OP160_EO_ATC_Tool_Presence_1,
    B7 => OP160_EO_ATC_Tool_Presence_2); // BYTE_AS_BIT

END_PROGRAM

// ---- POUs/Programs/OP160/OP160_Robo_Inputs.TcPOU
PROGRAM OP160_Robo_Inputs
VAR
	Robo_Enable_err: TON;
	Counter: R_TRIG;
	sampling_request_set :BOOL;
	sampling_count_reset : r_trig;
	Counter_reset        : BOOL;
END_VAR


// Safe to Pick
IF OP160_Moverpresent  THEN
	OP160_SI_Pick_Zone_Safe:=TRUE;
	 
	ELSE
		OP160_SI_Pick_Zone_Safe:=FALSE;
	END_IF
	
// Safe To Place
IF OP160_PartPicked THEN
	OP160_SI_Place_Zone_Safe:=TRUE;
	OP160_SI_Insert_Cylinder_Home := TRUE;
	ELSE
		OP160_SI_Place_Zone_Safe:=FALSE;
		OP160_SI_Insert_Cylinder_Home :=FALSE;
	END_IF
	
/// component status //	

	IF OP160_PartPicked THEN
       OP160_EI_Spare21 :=  op160_comp_rh_nok_to_rbt;
	   OP160_EI_Spare22  :=  op160_comp_lh_nok_to_rbt;
	END_IF   
	
////// robot go to pick ///////////////////////	
IF OP160_Moverpresent AND NOT OP160_PartPicked THEN
   OP160_EI_Rdy_Pick_QC:=TRUE;
   ELSE
   OP160_EI_Rdy_Pick_QC:=FALSE;
END_IF

/////// robot go to place /////////////////////////////
IF OP160_PartPicked AND ( op160_place_both_component_ok OR op160_go_to_place) THEN
	OP160_EI_Rdy_Place_QC:=TRUE;
ELSE
	OP160_EI_Rdy_Place_QC:=FALSE;
END_IF
	
///////////////////// robot go to rejection ///////////////
IF OP160_PartPicked AND ( op160_place_1_ok_1_nok OR op160_place_both_component_rej) THEN
   OP160_EI_Rdy_Place_Reject := TRUE;
ELSE
   OP160_EI_Rdy_Place_Reject := FALSE;
END_IF   


///////////////////////////////// production count ///////////////////////////////////////////////////
	
IF Counter_reset THEN
	Componenets_Produced:=0;
END_IF

IF Counter.Q AND NOT sampling_request_set THEN
	Componenets_Produced:=Componenets_Produced+1;
ELSIF Counter.Q AND  sampling_request_set THEN
	sampling_quantity := sampling_quantity+1;
END_IF

IF sampling_request  OR ((Componenets_Produced MOD sampling_interval)=0 AND (Componenets_Produced > 1)) THEN
   sampling_request_set:=TRUE; 
ELSIF NOT sampling_request OR sampling_quantity = sampling_request_qty THEN
   sampling_request_set:=FALSE;
END_IF

IF sampling_count_reset.Q THEN
   sampling_quantity:=0;
END_IF


sampling_count_reset(CLK:= sampling_request_set, Q=> );
Counter(CLK:=OP160_EO_QC_Place_Completed );

END_PROGRAM

// ---- POUs/Programs/OP120/OP120_Robo_Byte_Mapping.TcPOU
PROGRAM OP120_Robo_Byte_Mapping
VAR
	//Robo BYte Mapping Inputs
	OP120_Robo_IN_Byte1: BYTE_AS_BIT;
OP120_Robo_IN_6000_6007 AT %I*:BYTE;
OP120_Robo_IN_6008_6015 AT %I*:BYTE;
OP120_Robo_IN_6016_6023 AT %I*:BYTE;
OP120_Robo_IN_6024_6031 AT %I*:BYTE;
OP120_Robo_IN_6032_6039 AT %I*:BYTE;
OP120_Robo_IN_6040_6047 AT %I*:BYTE;
OP120_Robo_IN_6048_6055 AT %I*:BYTE;
OP120_Robo_IN_6056_6063 AT %I*:BYTE;
OP120_Robo_IN_6064_6071 AT %I*:BYTE;

//Robo Byte Mapping Out
OP120_Robo_Out_6000_6007 AT%Q*:BYTE;
OP120_Robo_Out_6008_6015 AT%Q*:BYTE;
OP120_Robo_Out_6016_6023 AT%Q*:BYTE;
OP120_Robo_Out_6024_6031 AT%Q*:BYTE;
OP120_Robo_Out_6032_6039 AT%Q*:BYTE;
OP120_Robo_Out_6040_6047 AT%Q*:BYTE;
OP120_Robo_Out_6048_6055 AT%Q*:BYTE;
OP120_Robo_Out_6056_6063 AT%Q*:BYTE;
OP120_Robo_Out_6064_6071 AT%Q*:BYTE;
//registerout

	OP120_Robo_IN_Byte2: BYTE_AS_BIT;
	OP120_Robo_IN_Byte3: BYTE_AS_BIT;
	OP120_Robo_IN_Byte4: BYTE_AS_BIT;
	OP120_Robo_IN_Byte5: BYTE_AS_BIT;
	OP120_Robo_IN_Byte6: BYTE_AS_BIT;
	OP120_Robo_IN_Byte7: BYTE_AS_BIT;
	OP120_Robo_IN_Byte8: BYTE_AS_BIT;
	OP120_Robo_Out_Byte1: BIT_AS_BYTE;
	OP120_Robo_Out_Byte2: BIT_AS_BYTE;
	OP120_Robo_Out_Byte3: BIT_AS_BYTE;
	OP120_Robo_Out_Byte4: BIT_AS_BYTE;
	OP120_Robo_Out_Byte5: BIT_AS_BYTE;
	OP120_Robo_Out_Byte6: BIT_AS_BYTE;
	OP120_Robo_Out_Byte7: BIT_AS_BYTE;
	OP120_Robo_Out_Byte8: BIT_AS_BYTE;
END_VAR

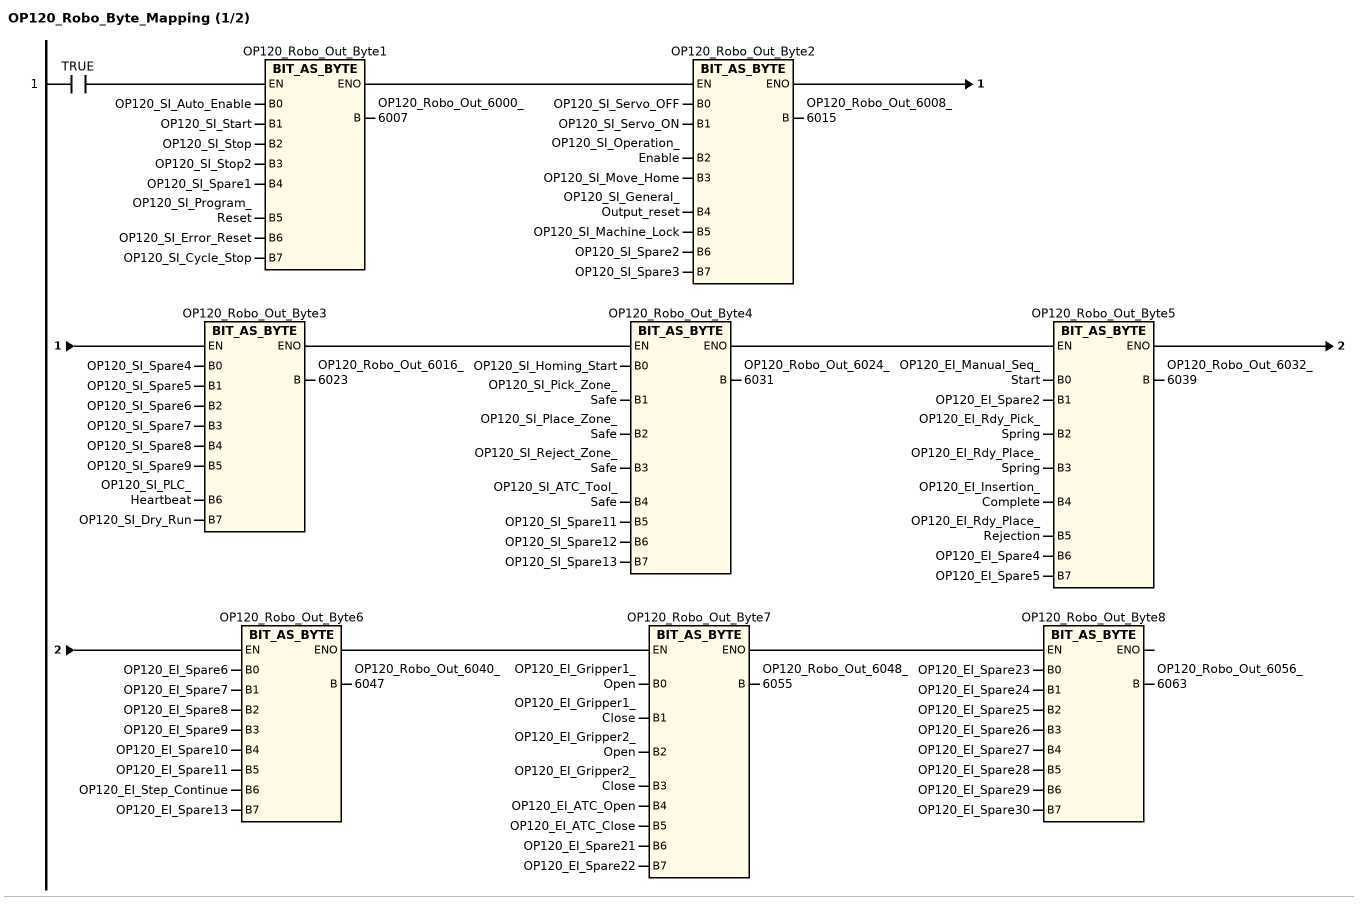
// NETWORK 1
OP120_Robo_Out_Byte1(
    B0 := OP120_SI_Auto_Enable,
    B1 := OP120_SI_Start,
    B2 := OP120_SI_Stop,
    B3 := OP120_SI_Stop2,
    B4 := OP120_SI_Spare1,
    B5 := OP120_SI_Program_Reset,
    B6 := OP120_SI_Error_Reset,
    B7 := OP120_SI_Cycle_Stop,
    B => OP120_Robo_Out_6000_6007); // BIT_AS_BYTE
OP120_Robo_Out_Byte2(
    B0 := OP120_SI_Servo_OFF,
    B1 := OP120_SI_Servo_ON,
    B2 := OP120_SI_Operation_Enable,
    B3 := OP120_SI_Move_Home,
    B4 := OP120_SI_General_Output_reset,
    B5 := OP120_SI_Machine_Lock,
    B6 := OP120_SI_Spare2,
    B7 := OP120_SI_Spare3,
    B => OP120_Robo_Out_6008_6015); // BIT_AS_BYTE
OP120_Robo_Out_Byte3(
    B0 := OP120_SI_Spare4,
    B1 := OP120_SI_Spare5,
    B2 := OP120_SI_Spare6,
    B3 := OP120_SI_Spare7,
    B4 := OP120_SI_Spare8,
    B5 := OP120_SI_Spare9,
    B6 := OP120_SI_PLC_Heartbeat,
    B7 := OP120_SI_Dry_Run,
    B => OP120_Robo_Out_6016_6023); // BIT_AS_BYTE
OP120_Robo_Out_Byte4(
    B0 := OP120_SI_Homing_Start,
    B1 := OP120_SI_Pick_Zone_Safe,
    B2 := OP120_SI_Place_Zone_Safe,
    B3 := OP120_SI_Reject_Zone_Safe,
    B4 := OP120_SI_ATC_Tool_Safe,
    B5 := OP120_SI_Spare11,
    B6 := OP120_SI_Spare12,
    B7 := OP120_SI_Spare13,
    B => OP120_Robo_Out_6024_6031); // BIT_AS_BYTE
OP120_Robo_Out_Byte5(
    B0 := OP120_EI_Manual_Seq_Start,
    B1 := OP120_EI_Spare2,
    B2 := OP120_EI_Rdy_Pick_Spring,
    B3 := OP120_EI_Rdy_Place_Spring,
    B4 := OP120_EI_Insertion_Complete,
    B5 := OP120_EI_Rdy_Place_Rejection,
    B6 := OP120_EI_Spare4,
    B7 := OP120_EI_Spare5,
    B => OP120_Robo_Out_6032_6039); // BIT_AS_BYTE
OP120_Robo_Out_Byte6(
    B0 := OP120_EI_Spare6,
    B1 := OP120_EI_Spare7,
    B2 := OP120_EI_Spare8,
    B3 := OP120_EI_Spare9,
    B4 := OP120_EI_Spare10,
    B5 := OP120_EI_Spare11,
    B6 := OP120_EI_Step_Continue,
    B7 := OP120_EI_Spare13,
    B => OP120_Robo_Out_6040_6047); // BIT_AS_BYTE
OP120_Robo_Out_Byte7(
    B0 := OP120_EI_Gripper1_Open,
    B1 := OP120_EI_Gripper1_Close,
    B2 := OP120_EI_Gripper2_Open,
    B3 := OP120_EI_Gripper2_Close,
    B4 := OP120_EI_ATC_Open,
    B5 := OP120_EI_ATC_Close,
    B6 := OP120_EI_Spare21,
    B7 := OP120_EI_Spare22,
    B => OP120_Robo_Out_6048_6055); // BIT_AS_BYTE
OP120_Robo_Out_Byte8(
    B0 := OP120_EI_Spare23,
    B1 := OP120_EI_Spare24,
    B2 := OP120_EI_Spare25,
    B3 := OP120_EI_Spare26,
    B4 := OP120_EI_Spare27,
    B5 := OP120_EI_Spare28,
    B6 := OP120_EI_Spare29,
    B7 := OP120_EI_Spare30,
    B => OP120_Robo_Out_6056_6063); // BIT_AS_BYTE

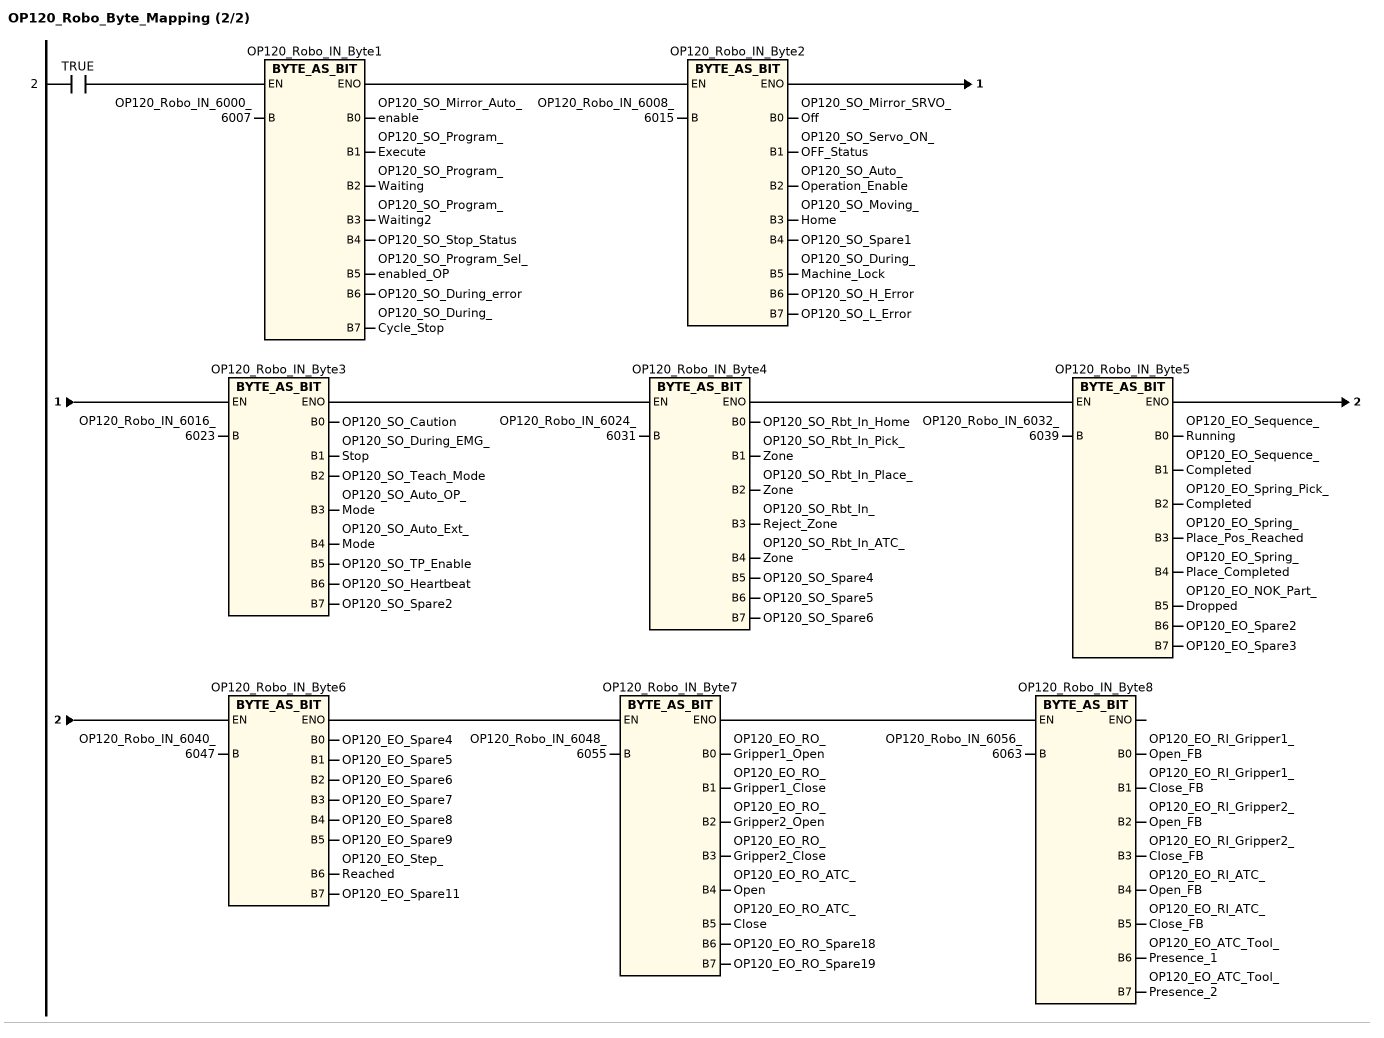
// NETWORK 2
OP120_Robo_IN_Byte1(
    B := OP120_Robo_IN_6000_6007,
    B0 => OP120_SO_Mirror_Auto_enable,
    B1 => OP120_SO_Program_Execute,
    B2 => OP120_SO_Program_Waiting,
    B3 => OP120_SO_Program_Waiting2,
    B4 => OP120_SO_Stop_Status,
    B5 => OP120_SO_Program_Sel_enabled_OP,
    B6 => OP120_SO_During_error,
    B7 => OP120_SO_During_Cycle_Stop); // BYTE_AS_BIT
OP120_Robo_IN_Byte2(
    B := OP120_Robo_IN_6008_6015,
    B0 => OP120_SO_Mirror_SRVO_Off,
    B1 => OP120_SO_Servo_ON_OFF_Status,
    B2 => OP120_SO_Auto_Operation_Enable,
    B3 => OP120_SO_Moving_Home,
    B4 => OP120_SO_Spare1,
    B5 => OP120_SO_During_Machine_Lock,
    B6 => OP120_SO_H_Error,
    B7 => OP120_SO_L_Error); // BYTE_AS_BIT
OP120_Robo_IN_Byte3(
    B := OP120_Robo_IN_6016_6023,
    B0 => OP120_SO_Caution,
    B1 => OP120_SO_During_EMG_Stop,
    B2 => OP120_SO_Teach_Mode,
    B3 => OP120_SO_Auto_OP_Mode,
    B4 => OP120_SO_Auto_Ext_Mode,
    B5 => OP120_SO_TP_Enable,
    B6 => OP120_SO_Heartbeat,
    B7 => OP120_SO_Spare2); // BYTE_AS_BIT
OP120_Robo_IN_Byte4(
    B := OP120_Robo_IN_6024_6031,
    B0 => OP120_SO_Rbt_In_Home,
    B1 => OP120_SO_Rbt_In_Pick_Zone,
    B2 => OP120_SO_Rbt_In_Place_Zone,
    B3 => OP120_SO_Rbt_In_Reject_Zone,
    B4 => OP120_SO_Rbt_In_ATC_Zone,
    B5 => OP120_SO_Spare4,
    B6 => OP120_SO_Spare5,
    B7 => OP120_SO_Spare6); // BYTE_AS_BIT
OP120_Robo_IN_Byte5(
    B := OP120_Robo_IN_6032_6039,
    B0 => OP120_EO_Sequence_Running,
    B1 => OP120_EO_Sequence_Completed,
    B2 => OP120_EO_Spring_Pick_Completed,
    B3 => OP120_EO_Spring_Place_Pos_Reached,
    B4 => OP120_EO_Spring_Place_Completed,
    B5 => OP120_EO_NOK_Part_Dropped,
    B6 => OP120_EO_Spare2,
    B7 => OP120_EO_Spare3); // BYTE_AS_BIT
OP120_Robo_IN_Byte6(
    B := OP120_Robo_IN_6040_6047,
    B0 => OP120_EO_Spare4,
    B1 => OP120_EO_Spare5,
    B2 => OP120_EO_Spare6,
    B3 => OP120_EO_Spare7,
    B4 => OP120_EO_Spare8,
    B5 => OP120_EO_Spare9,
    B6 => OP120_EO_Step_Reached,
    B7 => OP120_EO_Spare11); // BYTE_AS_BIT
OP120_Robo_IN_Byte7(
    B := OP120_Robo_IN_6048_6055,
    B0 => OP120_EO_RO_Gripper1_Open,
    B1 => OP120_EO_RO_Gripper1_Close,
    B2 => OP120_EO_RO_Gripper2_Open,
    B3 => OP120_EO_RO_Gripper2_Close,
    B4 => OP120_EO_RO_ATC_Open,
    B5 => OP120_EO_RO_ATC_Close,
    B6 => OP120_EO_RO_Spare18,
    B7 => OP120_EO_RO_Spare19); // BYTE_AS_BIT
OP120_Robo_IN_Byte8(
    B := OP120_Robo_IN_6056_6063,
    B0 => OP120_EO_RI_Gripper1_Open_FB,
    B1 => OP120_EO_RI_Gripper1_Close_FB,
    B2 => OP120_EO_RI_Gripper2_Open_FB,
    B3 => OP120_EO_RI_Gripper2_Close_FB,
    B4 => OP120_EO_RI_ATC_Open_FB,
    B5 => OP120_EO_RI_ATC_Close_FB,
    B6 => OP120_EO_ATC_Tool_Presence_1,
    B7 => OP120_EO_ATC_Tool_Presence_2); // BYTE_AS_BIT

END_PROGRAM

// ---- POUs/Programs/OP120/OP120_Robo_Inputs.TcPOU
PROGRAM OP120_Robo_Inputs
VAR
	Robo_Enable_err: TON;
	temp : ARRAY[1..500] OF BOOL;
	
END_VAR




// Safe to Pick
IF OperationEnable AND OP120_GVL.CR120_Lifting_Cyl.Position2  THEN
	OP120_SI_Pick_Zone_Safe:=TRUE;
	ELSE
		OP120_SI_Pick_Zone_Safe:=FALSE;
	END_IF
	
// Safe To Place
IF OperationEnable AND OP120_GVL.CR120_Horizontal_Push_Cyl.Position1 THEN
	OP120_IO_Tag_Link.OP120_SI_Place_Zone_Safe:=TRUE;
	ELSE
		OP120_IO_Tag_Link.OP120_SI_Place_Zone_Safe:=FALSE;
	END_IF
//Safe to Reject Zone
	
	IF OperationEnable AND TRUE THEN
		OP120_IO_Tag_Link.OP120_SI_Reject_Zone_Safe:=TRUE;
		ELSE
			OP120_IO_Tag_Link.OP120_SI_Reject_Zone_Safe:=FALSE;
		END_IF
// Safe to ATC Zone
IF OperationEnable THEN
	OP120_IO_Tag_Link.OP120_SI_ATC_Tool_Safe:=TRUE;
	ELSE
	OP120_IO_Tag_Link.OP120_SI_ATC_Tool_Safe:=FALSE;
	END_IF

//Ready to Pick
IF OP120_GVL.OP120_StartEnable AND OP120_GVL.CR120_Lifting_Cyl.Position2 AND OP120_GotoPick THEN 
	// AND CheckParkOK AND NOT  CheckParkNOK and (OP120_EI_Gripper1_Open AND  OP120_EI_Gripper2_Open OR temp [1])
   OP120_EI_Rdy_Pick_Spring :=TRUE;
ELSE
	OP120_IO_Tag_Link.OP120_EI_Rdy_Pick_Spring :=FALSE;
END_IF 

//REady to 	place

IF OP120_GVL.OP120_StartEnable AND OP120_GVL.CR120_Horizontal_Push_Cyl.Position1 AND OP120_MoverPresent  THEN //OP120_STN_ENABLE AND Part_Picked
	OP120_IO_Tag_Link.OP120_EI_Rdy_Place_Spring:=TRUE;
	ELSE
	OP120_IO_Tag_Link.OP120_EI_Rdy_Place_Spring:=FALSE;
END_IF

//Insertion Complete

IF OP120_GVL.OP120_StartEnable AND OP120_PartPushed THEN
	OP120_IO_Tag_Link.OP120_EI_Insertion_Complete:=TRUE;
ELSE
	OP120_IO_Tag_Link.OP120_EI_Insertion_Complete:=FALSE;
END_IF

END_PROGRAM

// ---- POU1/MAIN.TcPOU
PROGRAM MAIN
VAR
	brun 		AT %Q* : BOOL;
	bACK 		AT %Q* : BOOL;
	bSafety_OK  AT %I* : BOOL;
	bInit              : BOOL;
	Initialize		   : R_TRIG;
	Ack_Input		   : BOOL;
	Safety_Timer       : TON;	
	SafeOP_Timer	   : TON;
	EMG_Raise		   : R_TRIG;
	OP10A_Robo_State AT %I* : USINT;
	OP10B_Robo_State AT %I* : USINT;

	SERVO_TORQUE	AT %Q*	:UINT := 10000;
	
	ALL_LIGHTS_ON: BOOL;
	XTS_Lube_ON  : BOOL;
	
	All_Station_Auto_Mode     : BOOL;
	All_Station_Cycle_Start   : BOOL;
	All_Station_Cycle_Stop    : BOOL;
	Station_Ctrl_Temp         : BOOL;
	OP10_Lights_On			  : BOOL;
	tower_lamp_green_on       :BOOL;
	tower_lamp_red_on         :BOOL;
	tower_lamp_orange_on: BOOL;
	
	FB_Timer : FB_Time_Stamp_Maddy;
	Run_Time : STRING;
	Start_timer : BOOL;
	Stop_timer  : BOOL;
	Reset_timer : BOOL;
	Start_value : STRING;
	Stop_value  : STRING;
	Start_trig : R_TRIG;
	Stop_Trig  : R_TRIG;
	Reset_Trig : R_TRIG;
END_VAR


bACK			:= Pulse_Block.Q1Hz;

//Axis_Position_Bias();
O160_AUTOBAG_CNT_CMPLTD_Q707_4:=I10A_DRUM_OFF_ON_I714_2;
Initialize(CLK:=NOT bInit);
IF Initialize.Q THEN
	Ack_Input:=1;
	brun:=TRUE;
END_IF
SafeOP_Timer(IN:=Ack_Input,PT:=T#5S);
IF SafeOP_Timer.Q THEN
 bACK:=TRUE;
 Ack_Input:=0;
 bInit:=TRUE;
END_IF

Safety_Timer(IN:=bACK,PT:=T#500MS);
IF Safety_Timer.Q THEN
	bACK:=FALSE;
END_IF

EMG_Raise(CLK:=bSafety_OK , Q=> );
IF EMG_Raise.Q THEN
   bACK:=TRUE;
END_IF

RFID();
Error();
OP10_MAIN();
OP20_MAIN();
OP30_MAIN();
OP40_MAIN();
OP50_MAIN();
OP60_MAIN();
OP70_MAIN();
OP80_MAIN();
OP90_MAIN();
OP110_MAIN();
OP120_MAIN();
OP130_MAIN();
OP140_MAIN();
OP160_MAIN();
IO_Diag();
IO_OP10_PANEL();
IO_OP10A_10B_JB();
Master1_IO_Map();
MASTER2_IO_Map();
OP90_MP_IO();
OP90_MASTER3_IO();
OP90_JB_IO();
OP160_MP_IO();
OP160_MASTER4_IO();
OP120_JB_IO();
OP150_Main();
MAIN_1();
EtherCatDiag();
//MOdeselection From HMI
IF (HMI_AutoMode AND NOT HMI_ManualMOde AND NOT HMI_StepMode) THEN
		FB_MODE_BLOCK.ModeWord:=1;
	ELSIF (NOT HMI_AutoMode AND HMI_ManualMOde AND NOT HMI_StepMode) THEN
		FB_MODE_BLOCK.ModeWord:=2;
	ELSIF  (NOT HMI_AutoMode AND NOT HMI_ManualMOde AND HMI_StepMode) THEN
		FB_MODE_BLOCK.ModeWord:=3;
    ELSE   
		FB_MODE_BLOCK.ModeWord:=0;
END_IF

Servo_safety     := bSafety_OK;
OperationEnable  := bSafety_OK;

IF OperationEnable THEN
	Servo_Enable:=TRUE;
ELSE
	Servo_Enable:=FALSE;
END_IF

FB_MODE_BLOCK(
	ModeWord:= , 
	HomeConditionOK:= ALL_STN_IN_HOME, 
	OperationEnable:= bSafety_OK , 
	StartPB:= START_PB, 
	SafetyAndNOError:= bSafety_OK AND NOT ERROR_ACTIVE, 
	ModeAck:= TRUE , 
	HomingINProgress:= , 
	TempHomeOK:= , 
	ResetPB:= , 
	AutoSelected=>AUTO_SELECTED , 
	ManualSelected=> MANUAL_SELECTED, 
	StepSelected=> STEP_SELECTED, 
	ModeSelAck_Indication=> , 
	StatusDisplay=> , 
	AutoRunning:=AUTO_RUNNING , 
	StepRunning:=STEP_RUNNING , 
	StartEnable:=START_ENABLE , 
	MachineStop:=MACHINE_STOP);
	
Pulse_Block(
	Q10Hz=> , 
	Q5Hz=> , 
	Q2_5Hz=> , 
	Q2Hz=> , 
	Q1_25Hz=> , 
	Q2Hz=> , 
	Q0_625Hz=> , 
	Q0_5Hz=> );	
	
IF ALL_LIGHTS_ON THEN				
		O30_CAM_LGHT1_ON_Q305_1                  :=1;
		O30_CAM_LGHT2_ON_Q305_2                  :=1;
		O50_CAM_LGHT1_ON_Q306_3                  :=1;
		O50_CAM_LGHT2_ON_Q306_4                  :=1;
		O70_CAM_LGHT1_ON_Q307_6                  :=1;
		O70_CAM_LGHT2_ON_Q307_7                  :=1;
		O90_VISN_LGHT1_ON_Q400_0                 :=1;
		O90_VISN_LGHT2_ON_Q400_1                 :=1;
		O120_VISN_LGHT1_ON_Q402_4                :=1;
		O120_VISN_LGHT2_ON_Q402_5                :=1;
		O150_VISN_LGHT_ON_Q706_6                 :=1;
		O160_CHECKER_LGHT_ON_Q707_1              :=1;
ELSE		
		O30_CAM_LGHT1_ON_Q305_1                  :=0;
		O30_CAM_LGHT2_ON_Q305_2                  :=0;
		O50_CAM_LGHT1_ON_Q306_3                  :=0;
		O50_CAM_LGHT2_ON_Q306_4                  :=0;
		O70_CAM_LGHT1_ON_Q307_6                  :=0;
		O70_CAM_LGHT2_ON_Q307_7                  :=0;
		O90_VISN_LGHT1_ON_Q400_0                 :=0;
		O90_VISN_LGHT2_ON_Q400_1                 :=0;
		O120_VISN_LGHT1_ON_Q402_4                :=0;
		O120_VISN_LGHT2_ON_Q402_5                :=0;
		O150_VISN_LGHT_ON_Q706_6                 :=0;
		O160_CHECKER_LGHT_ON_Q707_1              :=0;	
END_IF

IF OP10_Lights_On THEN
		O10A_BDY_EMPT_CAM_LGHT1_ON_Q301_0        :=1; 
		O10A_BDY_EMPT_CAM_LGHT2_ON_Q301_1        :=1;
//		O10A_FIRTREE_ORING_CAM_LGHT1_ON_Q301_2   :=1;
//		O10A_FIRTREE_ORING_CAM_LGHT2_ON_Q301_3   :=1;
		O10A_ORING_CAM_LGHT1_ON_Q301_4           :=1;
		O10A_ORING_CAM_LGHT2_ON_Q301_5           :=1;
//		O10A_FIRTREE_ORING_CAMBAR_LGHT1_ON_Q301_6:=1;
//		O10B_FIRTREE_ORING_CAM_LGHT1_ON_Q303_2   :=1;
//		O10B_FIRTREE_ORING_CAM_LGHT2_ON_Q303_3   :=1;
		O10B_ORING_CAM_LGHT1_ON_Q303_4           :=1;
		O10B_ORING_CAM_LGHT2_ON_Q303_5           :=1;
//		O10B_FIRTREE_ORING_CAMBAR_LGHT1_ON_Q303_6:=1;
ELSE
		O10A_BDY_EMPT_CAM_LGHT1_ON_Q301_0        :=0; 
		O10A_BDY_EMPT_CAM_LGHT2_ON_Q301_1        :=0;
		O10A_FIRTREE_ORING_CAM_LGHT1_ON_Q301_2   :=0;
		O10A_FIRTREE_ORING_CAM_LGHT2_ON_Q301_3   :=0;
		O10A_ORING_CAM_LGHT1_ON_Q301_4           :=0;
		O10A_ORING_CAM_LGHT2_ON_Q301_5           :=0;
		O10A_FIRTREE_ORING_CAMBAR_LGHT1_ON_Q301_6:=0;
		O10B_FIRTREE_ORING_CAM_LGHT1_ON_Q303_2   :=0;
		O10B_FIRTREE_ORING_CAM_LGHT2_ON_Q303_3   :=0;
		O10B_ORING_CAM_LGHT1_ON_Q303_4           :=0;
		O10B_ORING_CAM_LGHT2_ON_Q303_5           :=0;
		O10B_FIRTREE_ORING_CAMBAR_LGHT1_ON_Q303_6:=0;	
END_IF
		
		
IF XTS_Lube_ON THEN
	O10_XTS_GREASE_VALVE_ON_Q300_0:=Pulse_Block.Q0_5Hz;
ELSE	
	O10_XTS_GREASE_VALVE_ON_Q300_0:=0;
END_IF
		
O150_BARLIGHT_OP1_Q706_7 :=	Pulse_Block.Q2_5Hz;
O150_BARLIGHT_OP2_Q707_0 := Pulse_Block.Q1Hz;	
                                                      
O10_TWR_LMP_RD_Q302_5   := Pulse_Block.Q1Hz AND tower_lamp_green_on;                         
O10_TWR_LMP_GN_Q302_6   := Pulse_Block.Q1Hz AND tower_lamp_red_on;                        
O10_TWR_LMP_YELW_Q302_7 := Pulse_Block.Q1Hz AND tower_lamp_orange_on;
O120_TWR_LMP_GN_Q403_1   := Pulse_Block.Q1Hz AND tower_lamp_green_on;
O120_TWR_LMP_YELW_Q403_2 := Pulse_Block.Q1Hz AND tower_lamp_orange_on ;
O120_TWR_LMP_RD_Q403_0   := Pulse_Block.Q1Hz AND tower_lamp_red_on;	

O10_BARLIGHT_OP1_Q300_6  := Pulse_Block.Q1Hz;
O10_BARLIGHT_OP2_Q300_7  := Pulse_Block.Q1_25Hz;	

IF NOT OperationEnable THEN
	OP20_ErrorActive:=1;
	OP30_ErrorActive:=1;
	OP40_ErrorActive:=1;
	OP50_ErrorActive:=1;
	OP60_ErrorActive:=1;
	OP70_ErrorActive:=1;
	OP80_ErrorActive:=1;
	OP110_ErrorActive:=1;
	OP120_ErrorActive:=1;
	OP130_ErrorActive:=1;
	OP140_ErrorActive:=1;
	OP160_ErrorActive:=1;
END_IF

IF AUTO_WITH_XTS AND Station_Ctrl_Temp THEN

	IF All_Station_Auto_Mode THEN
		OP20_HMI_AutoMode:=1;
		OP30_HMI_AutoMode:=1;
		OP40_HMI_AutoMode:=1;
		OP50_HMI_AutoMode:=1;
		OP60_HMI_AutoMode:=1;
		OP70_HMI_AutoMode:=1;
		OP80_HMI_AutoMode:=1;	
		OP110_HMI_AutoMode:=1;	
        OP120_HMI_AutoMode:=1;
		OP130_HMI_AutoMode:=1;	
	//	OP140_HMI_AutoMode:=1;
        OP160_HMI_AutoMode:=1;			
	END_IF
	IF All_Station_Cycle_Start THEN
		OP20_HMI_CycleStart	:=1;
		OP30_HMI_Cycle_Start:=1;
		OP40_HMI_Cycle_Start:=1;
		OP50_HMI_Cycle_Start:=1;
		OP60_HMI_CycleStart	:=1;
		OP70_HMI_Cycle_Start:=1;
		OP80_HMI_CycleStart	:=1;
		OP110_HMI_CycleStart:=1;
		OP120_HMI_CycleStart_PB:=1;
		OP130_HMI_CycleStart:=1;
	//	OP140_HMI_CycleStart:=1;
		OP160_HMI_CycleStart:=1;
	ELSE
		OP20_HMI_CycleStart	:=0;
		OP30_HMI_Cycle_Start:=0;
		OP40_HMI_Cycle_Start:=0;
		OP50_HMI_Cycle_Start:=0;
		OP60_HMI_CycleStart	:=0;
		OP70_HMI_Cycle_Start:=0;
		OP80_HMI_CycleStart	:=0;
		OP110_HMI_CycleStart:=0;	
		OP120_HMI_CycleStart_PB:=0;
		OP130_HMI_CycleStart:=0;
	//	OP140_HMI_CycleStart:=0;
		OP160_HMI_CycleStart:=0;		
	END_IF
	IF All_Station_Cycle_Stop THEN
		 OP20_Stop_Request  :=1;
 		 OP30_Stop_Request  :=1;
 		 OP40_Stop_Request  :=1;
 		 OP50_Stop_Request  :=1;
 		 OP60_Stop_Request  :=1;
 		 OP70_Stop_Request  :=1;
 		 OP80_Stop_Request  :=1;
 		 OP110_Stop_Request :=1;
		 OP120_Machine_Stop :=1;
		 OP130_Machine_Stop	:=1;
		// OP140_Machine_Stop :=1;
		 OP160_Machine_Stop	:=1;
	ELSE
		 OP20_Stop_Request  :=0;
 		 OP30_Stop_Request  :=0;
 		 OP40_Stop_Request  :=0;
 		 OP50_Stop_Request  :=0;
 		 OP60_Stop_Request  :=0;
 		 OP70_Stop_Request  :=0;
 		 OP80_Stop_Request  :=0;
 		 OP110_Stop_Request :=0;
		 OP120_Machine_Stop :=0;
		 OP130_Machine_Stop	:=0;
		// OP140_Machine_Stop :=0;
		 OP160_Machine_Stop	:=0;	 
	END_IF
END_IF	


////// tower lamp ////////////////////
IF OP10A_AUTO_RUNNING AND  OP160_AutoRunning AND  OP140_AutoRunning AND 
   OP130_AutoRunning AND OP110_AutoRunning AND OP120_AutoRunning  AND 
   OP90_AUTO_RUNNING AND OP80_AutoRunning AND OP70_AutoRunning AND 
   OP60_AutoRunning AND  OP50_AutoRunning AND OP40_AutoRunning AND 
   OP30_AutoRunning AND OP20_AutoRunning THEN
   tower_lamp_green_on := TRUE;
   tower_lamp_red_on   := FALSE;
   tower_lamp_orange_on:=FALSE;	
END_IF

IF NOT (OP160_AutoRunning AND  OP140_AutoRunning AND  OP130_AutoRunning AND 
        OP10A_AUTO_RUNNING AND OP110_AutoRunning AND OP120_AutoRunning AND
        OP90_AUTO_RUNNING AND OP80_AutoRunning AND OP70_AutoRunning AND
        OP60_AutoRunning AND OP50_AutoRunning AND OP40_AutoRunning AND
        OP30_AutoRunning AND OP20_AutoRunning) THEN
	    tower_lamp_green_on :=FALSE ;
	    tower_lamp_red_on   := FALSE;
        tower_lamp_orange_on:=TRUE;	
END_IF

IF  OP10A_ERR OR OP10B_ERR OR OP110_ErrorActive OR OP120_ErrorActive OR OP130_ErrorActive OR OP140_ErrorActive
    OR OP160_ErrorActive OR OP90_ERR OR OP80_ErrorActive OR OP70_ErrorActive OR OP60_ErrorActive OR
	OP50_ErrorActive OR OP40_ErrorActive OR OP30_ErrorActive OR OP20_ErrorActive THEN
        tower_lamp_green_on :=FALSE ;
		tower_lamp_red_on   := TRUE;
		tower_lamp_orange_on:=FALSE;	
END_IF			
		
//////////////////

fbTime();

logTimer( IN := fbTime.bValid );
IF logTimer.Q THEN
    logTimer( IN := FALSE );
	logTimer( IN := fbTime.bValid );
    ADSLOGSTR( ADSLOG_MSGTYPE_HINT OR ADSLOG_MSGTYPE_LOG, 'Local System Time:%s', SYSTEMTIME_TO_STRING(fbTime.systemTime));
END_IF	

	wYear	:= fbTime.systemTime.wYear;
	wMonth	:= fbTime.systemTime.wMonth;
	wDate   := fbTime.systemTime.wDay;
	wHour	:= fbTime.systemTime.wHour;
	wMinute := fbTime.systemTime.wMinute;
	wSecond := fbTime.systemTime.wSecond;
	wMillisec:= fbTime.systemTime.wMilliseconds;
	
FB_Timer(
	Start:= , 
	Stop:= , 
	Running_Timer=> Run_Time, 
	Time_Difference_ms=> , 
	Time_Struct:=fbTime.systemTime );	
	
Start_trig(CLK:=Start_timer);	
Stop_trig(CLK :=Stop_timer);
Reset_Trig(CLK:=Reset_timer);	
	
IF Start_trig.Q THEN
	Start_value:=Run_Time;
END_IF
IF Stop_trig.Q THEN
	Stop_value:=Run_Time;
END_IF
IF Reset_Trig.Q THEN
	Start_value:=' ';
	Stop_value:=' ';
END_IF

END_PROGRAM

// ---- POU1/FB_Time_Stamp_Maddy.TcPOU
FUNCTION_BLOCK FB_Time_Stamp_Maddy
VAR_INPUT
	Start       : BOOL;
	Stop		: BOOL;
END_VAR
VAR_OUTPUT
	Running_Timer 		: STRING;
	Time_Difference_ms  : WORD; 
END_VAR
VAR_IN_OUT
	Time_Struct : TIMESTRUCT;
END_VAR
VAR
	Txt1 : STRING;
	Colon : STRING :=':';
	Txt2 : STRING;
	Txt3 : STRING;
	Txt4 : STRING;
	Txt5 : STRING;
	Txt6 : STRING;
	Start_trig :R_TRIG;
	Stop_trig  :R_TRIG;
END_VAR

VAR PERSISTENT
	START_TIME : TIMESTRUCT;
	STOP_TIME  : TIMESTRUCT;
END_VAR

Start_trig(CLK:=Start );
Stop_trig(CLK:=Stop );
IF Start_trig.Q THEN
	START_TIME:=Time_Struct;
END_IF
IF Stop_trig.Q THEN
	STOP_TIME:=Time_Struct;
END_IF

Txt1:=CONCAT(WORD_TO_STRING(Time_Struct.wHour),Colon);
Txt2:=CONCAT(Txt1,WORD_TO_STRING(Time_Struct.wMinute));
Txt3:=CONCAT(Txt2,Colon);
Txt4:=CONCAT(Txt3,WORD_TO_STRING(Time_Struct.wSecond));
Txt5:=CONCAT(Txt4,Colon);
Txt6:=CONCAT(Txt5,WORD_TO_STRING(Time_Struct.wMilliseconds));

Running_Timer:=Txt6;

END_FUNCTION_BLOCK

// ---- POU1/RFID.TcPOU
PROGRAM RFID
VAR
   in_1 AT %I*: ARRAY[0..63] OF BYTE;
   out_1 AT %Q*: ARRAY[0..63] OF BYTE;

   in_2 AT %I*: ARRAY[0..63] OF BYTE;
   out_2 AT %Q*: ARRAY[0..63] OF BYTE;   
   
   data_1 : HeadData;
   state_1 : head1;
   channel_1 : Memory;
   write_1 , quit_1 , restart_1 , finish_1: BOOL;
   busy_1,done_1,notag_1,error_1 : BOOL;
   status_1,counter_1 : BYTE;
   ident_1: FB_RFID;
   read_1: BOOL;
   
   data_2 : HeadData;
   state_2 : head1;
   channel_2 : Memory;
   write_2 , quit_2 , restart_2 , finish_2: BOOL;
   busy_2,done_2,notag_2,error_2 : BOOL;
   status_2,counter_2 : BYTE;
   ident_2: FB_RFID;
   read_2: BOOL;


END_VAR

ident_1(
	I_T_Timeout:=T#10S , 
	I_b_Head1SingleEnhanced:= , 
	I_b_Head1DataFixcode:= , 
	I_b_Head1SpecialFixcode:= , 
	I_b_Head1SpecialCommand:= , 
	I_b_Head1Read:= read_1 , 
	I_b_Head1Write:= write_1 , 
	I_b_Head1Quit:= quit_1, 
	I_i_Head1WordNum:= 1, 
	I_w_Head1WordAddress:=  , 
	I_w_Head1TagType:= 16#3033 , 
	HwIn:= in_1, 
	IO_b_SetRestart:= restart_1, 
	IO_b_InitFinish:= finish_1, 
	Head1Data:= data_1 ,
	head1:= state_1,
	Memory:= channel_1 , 
	O_b_Head1Busy=> busy_1, 
	O_b_Head1Done=> done_1, 
	O_b_Head1NoDataCarrier=>notag_1 , 
	O_b_Head1Error=> error_1, 
	O_B_Head1Status=> status_1, 
	O_B_Head1ReplyCounter=> counter_1, 
	HwOut=> out_1 );

ident_2(
	I_T_Timeout:=T#10S , 
	I_b_Head1SingleEnhanced:= , 
	I_b_Head1DataFixcode:= , 
	I_b_Head1SpecialFixcode:= , 
	I_b_Head1SpecialCommand:= , 
	I_b_Head1Read:= read_2 , 
	I_b_Head1Write:= write_2 , 
	I_b_Head1Quit:= quit_2, 
	I_i_Head1WordNum:= 1, 
	I_w_Head1WordAddress:=  , 
	I_w_Head1TagType:= 16#3033 , 
	HwIn:= in_2, 
	IO_b_SetRestart:= restart_2, 
	IO_b_InitFinish:= finish_2, 
	Head1Data:= data_2 ,
	head1:= state_2,
	Memory:= channel_2 , 
	O_b_Head1Busy=> busy_2, 
	O_b_Head1Done=> done_2, 
	O_b_Head1NoDataCarrier=>notag_2 , 
	O_b_Head1Error=> error_2, 
	O_B_Head1Status=> status_2, 
	O_B_Head1ReplyCounter=> counter_2, 
	HwOut=> out_2 );


//IF notag_1 OR error_1 THEN
//	restart_1:=TRUE;
//ELSE
//    restart_1:=FALSE;
//END_IF	
//
//IF notag_2 OR error_2 THEN
//	restart_2:=TRUE;
//ELSE
//    restart_2:=FALSE;
//END_IF

END_PROGRAM

// ---- FB/RFID/FB_RFID.TcPOU
FUNCTION_BLOCK FINAL FB_RFID
VAR_INPUT
I_T_Timeout: 						TIME;
I_b_Head1SingleEnhanced:	 		BOOL;
I_b_Head1DataFixcode:				BOOL;
I_b_Head1SpecialFixcode:			BOOL;
I_b_Head1SpecialCommand:			BOOL;
I_b_Head1Read:						BOOL;
I_b_Head1Write:						BOOL;
I_b_Head1Quit:						BOOL;
I_i_Head1WordNum:					INT;
I_w_Head1WordAddress:				WORD;
I_w_Head1TagType:					WORD;
HwIn:								ARRAY [0..63] OF BYTE;
END_VAR
VAR_IN_OUT
IO_b_SetRestart:					BOOL;
IO_b_InitFinish:					BOOL;
Head1Data:							HeadData;
head1:								Head1;
Memory:								Memory;
END_VAR
VAR_OUTPUT
O_b_Head1Busy:						BOOL;
O_b_Head1Done:						BOOL;
O_b_Head1NoDataCarrier:				BOOL;
O_b_Head1Error:						BOOL;
O_B_Head1Status:					BYTE;
O_B_Head1ReplyCounter:				BYTE;	
HwOut:								ARRAY [0..63] OF BYTE;
END_VAR
VAR
state_init:							INT;
state_cmd1:							INT;
i:									INT;
RTRIG_Read1:						R_TRIG;
RTRIG_Write1:						R_TRIG;
RTRIG_Quit1:						R_TRIG;
RTRIG_SpecialCommand1:				R_TRIG;
RTRIG_SetRestart:					R_TRIG;

Head_1_InData: 						ARRAY [0..63] OF BYTE;
Head_1_OutData:						ARRAY [0..63] OF BYTE;
Watchdog1:							TON;
temp								: BOOL;

END_VAR


(* Receive complete Input-Telegram from IdentControl each cycle *)
 Memory.Memory := HwIn; 


(* Check telegram *)

    
    IF Memory.OldReplyCounter <> Memory.Memory[3] THEN (* New telegram available *)
        Memory.Headnumber := SHR(Memory.Memory[1] AND 16#E, 1); (* Get channel number *)
        Memory.Togglebit := (Memory.Memory[1] AND 16#1); (* Get togglebit *)
        Memory.OldCommandIn := Memory.Memory[0];
        Memory.OldChannelIn := Memory.Memory[1];
        Memory.OldStatus := Memory.Memory[2];
        Memory.OldReplyCounter := Memory.Memory[3];
         IF Memory.Headnumber = 1 THEN
			MEMCPY( srcAddr:=ADR(Memory.Memory[0]),destAddr:=ADR(Head_1_InData[0])  , n:=SIZEOF( Memory.Memory));
			MEMCPY( srcAddr:=ADR(Head_1_InData[4]),  destAddr:=ADR(Head1Data.ReadData[0]), n:=SIZEOF ( Head_1_InData));
            Head1.NewData := TRUE;
 		  END_IF;
      
     END_IF;
 

 
(* Define inputs as rising edges *)
RTRIG_SetRestart(CLK := IO_b_SetRestart);
RTRIG_Read1(CLK := I_b_Head1Read);
RTRIG_Write1(CLK := I_b_Head1Write);
RTRIG_Quit1(CLK := I_b_Head1Quit);
RTRIG_SpecialCommand1(CLK := I_b_Head1SpecialCommand);

(* Acknowledge rising edge *)
IF RTRIG_Read1.Q THEN
    Head1.SaveRead := TRUE;
ELSIF RTRIG_Write1.Q THEN
    Head1.SaveWrite := TRUE;
ELSIF RTRIG_Quit1.Q THEN
    Head1.SaveQuit := TRUE;
ELSIF RTRIG_SpecialCommand1.Q THEN
    Head1.SaveSpecialCommand := TRUE;
END_IF;

IF RTRIG_SetRestart.Q THEN
    Head1.ExistTC := FALSE;
    Head1.NotExist := FALSE;
    Head1.Done := FALSE;
    O_b_Head1Done := FALSE;
    Head1.Error := FALSE;
    O_b_Head1Error := FALSE;
    Head1.Busy := FALSE;
    O_b_Head1Busy := FALSE;
    Head1.NoDataCarrier := FALSE;
    O_b_Head1NoDataCarrier := FALSE;
    Head1.SglCommandActive := FALSE;
    Head1.EnhCommandActive := FALSE;
    Head1.NewData := FALSE;
    Head1.TimeoutActive := FALSE;
    Head1.TimeoutOccurred := FALSE;
    Head1.TransfToHead := FALSE;
    Head1.SendOK := FALSE;
    Head1.Execute := FALSE;
    Head1.ReceiveOK := FALSE;
    Head1.SaveRead := FALSE;
    Head1.SaveWrite := FALSE;
    Head1.SaveQuit := FALSE;
    Head1.SaveSpecialCommand := FALSE;
    
    state_init := 1;
    state_cmd1 := 0;
    IO_b_InitFinish := FALSE;
END_IF;

(* ******************** Initialize routine ******************** *)
CASE state_init OF
        
    0:  (* ********************** Idle state ******************* *)
		;   
    1:  (* ********************** Initialize variables  ******************* *)
        
        (* Clear OutData array *)
        FOR i := 0 TO 63 BY 1 DO               //overwrite output data field of head 1
            Head_1_OutData[i] := 16#0;        //new in V2.1
        END_FOR;
        
        FOR i := 0 TO 59 BY 1 DO               //overwrite Write Data field of head 1
            Head1Data.WriteData[i] := 16#0;
        END_FOR;
        
        (* Clear InData array *)
        FOR i := 0 TO 63 BY 1 DO               //overwrite input data field of head 1
            Head_1_InData[i] := 16#0;         //new in V2.1
            Memory.Memory[i] := 16#0;         //cverwrite Memory Input data field
        END_FOR;
        
        FOR i := 0 TO 59 BY 1 DO
             Head1Data.ReadData[i] := 16#0;   //overwrite Read Data field of head 1
        END_FOR;
        
        
        state_init := state_init + 1;   (* Go to next state *)
        
        
    2: (* ***************** Send Change Tag Command For Channel 1 *************** *)
        
        (* Init OUTPUT Array with command *)
        Head_1_OutData[0] := 16#04;    (*Command: Change Tag*)
        Head_1_OutData[1] := 16#02;
        Head_1_OutData[2] := WORD_TO_BYTE(SHR(I_w_Head1TagType, 8));
        Head_1_OutData[3] := WORD_TO_BYTE(I_w_Head1TagType);
        
        Head1.Busy := TRUE;
        O_b_Head1Busy := TRUE;
        Head1.Done := FALSE;
        O_b_Head1Done := FALSE;
        Head1.TimeoutActive := TRUE;
        
        (* Invert togglebit to inform PLC, that a new telegram is available *)
        IF Memory.Togglebit <> 1 THEN
            Head_1_OutData[1] := Head_1_OutData[1] OR 16#1;
        ELSE
            Head_1_OutData[1] := Head_1_OutData[1] AND 16#FE;
        END_IF;
        
        HwOut:=Head_1_OutData ; (* Write on BUS *)  (* Write on BUS *)
     
           
            state_init := state_init + 1; (* Go to next state *)
        
        
        
    3: (* ******************** Wait for CT ************************ *)
        IF Head1.NewData THEN
            
            Head1.NewData := FALSE;
            O_B_Head1Status := Head_1_InData[2];
            O_B_Head1ReplyCounter := Head_1_InData[3];
            
            (* Antenna OK *)
            IF Head_1_InData[2] = 16#0 THEN
                Head1.ExistTC := TRUE;
                Head1.NotExist := FALSE;
            END_IF;
            (* Antenna not OK *)
            IF Head_1_InData[2] = 16#6 THEN
                Head1.ExistTC := FALSE;
                Head1.NotExist := TRUE;
            END_IF;
            
            (* Error *)
            IF Head_1_InData[2] = 16#4
                OR Head_1_InData[2] = 16#7
                OR Head_1_InData[2] = 16#9 THEN
                Head1.ExistTC := FALSE;
                Head1.NotExist := FALSE;
                Head1.Error := TRUE;
                O_b_Head1Error := TRUE;
            END_IF;
            
            (* Done *)
            IF Head_1_InData[2] <> 16#FF THEN
                Head1.Busy := FALSE;
                O_b_Head1Busy := FALSE;
                Head1.Done := TRUE;
                O_b_Head1Done := TRUE;
                Head1.TimeoutActive := FALSE;
                state_init := state_init + 1; (* Go to next state *)
            END_IF;
        END_IF;
        
    4:  (* Initialization finished *)
        IF (Head1.ExistTC OR Head1.NotExist) THEN
            IO_b_InitFinish := TRUE;
           // SetRestart := False;           //new in V2.1; Reset SetRestart from inside FB
        END_IF;
END_CASE;

(* ******************** Function block ready ******************** *)
IF IO_b_InitFinish THEN
(* ********** Commands Channel 1 ********** *)
    IF NOT Head1.Execute THEN
        
        (* ***** Quit ***** *)
        IF Head1.SaveQuit THEN
            Head_1_OutData[0] := 16#2;
            
            Head1.EnhCommandActive := FALSE;
            Head1.Execute := TRUE;
            state_cmd1 := 1;
        END_IF;
        
        (* ***** Single Read Words ***** *)
        IF Head1.SaveRead AND NOT I_b_Head1DataFixcode AND NOT I_b_Head1SingleEnhanced AND NOT I_b_Head1SpecialFixcode THEN
            Head_1_OutData[0] := 16#10;
            Head_1_OutData[1] := WORD_TO_BYTE((INT_TO_WORD(SHL(I_i_Head1WordNum, 4)) OR 16#2));
            Head_1_OutData[2] := WORD_TO_BYTE(SHR( I_w_Head1WordAddress AND 16#FF00,8));
            Head_1_OutData[3] := WORD_TO_BYTE(I_w_Head1WordAddress);
            
            Head1.SglCommandActive := TRUE;
            Head1.EnhCommandActive := FALSE;
            Head1.Execute := TRUE;
            state_cmd1 := 1;
        END_IF;
        
        (* ***** Single Read Fixcode ***** *)
        IF Head1.SaveRead AND I_b_Head1DataFixcode AND NOT I_b_Head1SingleEnhanced AND NOT I_b_Head1SpecialFixcode THEN
            Head_1_OutData[0] := 16#01;
            Head_1_OutData[1] := 16#02;
            
            Head1.SglCommandActive := TRUE;
            Head1.EnhCommandActive := FALSE;
            Head1.Execute := TRUE;
            state_cmd1 := 1;
        END_IF;
        
